(* CODESYS project bkp_29_07_24_VER_3_17.project
   Project Profile: Single

Project tree, tasks and I/O mapping:
  Device : NX3010, Altus S.A., order no. NX3010, version 1.2.1.233
    application Application
      libraries: NX5001 Diagnostic Structs, * (WAA); NX1005 Diagnostic Structs, * (WAA); NX2020 Diagnostic Structs, * (WAA); NX5000 Diagnostic Structs, * (WAA); NX6020 Diagnostic Structs, * (Manufacturer); Util, 3.5.1.0 (System); NextoStandard, 1.1.0.26 (WAA); LibDataTypes, 1.0.0.0 (Manufacturer); NX3010 Diagnostic Structs, 1.1.0.2 (WAA); NX2001 Diagnostic Structs, 1.0.0.5 (WAA); NX1001 Diagnostic Structs, 1.0.0.4 (WAA); NX6000 Diagnostic Structs, 0.0.0.2 (WAA); NX6010 Diagnostic Structs, 0.0.0.5 (Manufacturer); NX6100 Diagnostic Structs, 0.0.0.2 (WAA); NX4000 Diagnostic Structs, 1.0.0.0 (WAA); NXModbus Diagnostic Structs, 1.0.0.4 (WAA); NextoPID, 1.0.0.9 (WAA); Standard, 3.5.15.0 (System); Standard, * (System); SysTime, 3.5.9.0 (System); CAA File, 3.5.12.0 (CAA Technical Workgroup); CAA Callback Extern, 3.5.11.0 (CAA Technical Workgroup); CAA Memory Block Manager Extern, 3.5.7.0 (CAA Technical Workgroup); CAA Ressource Manager Extern, 3.5.11.0 (CAA Technical Workgroup); CAA Types Extern, 3.5.10.0 (CAA Technical Workgroup)
      task Configuration (cyclic, interval 9000 µs, priority 4) calls Configuration.EtherCAT_Task [Configuration.EtherCAT_Task]
      task MainTask (cyclic, interval 100 ms, priority 13, watchdog 1000 ms x 1) calls MainPrg
      task ATModbusMODBUS_Server (cyclic, interval 50 ms, priority 16) calls MODBUS_Server_Instance.Task
      task ATModbusMODBUS_RTU_Master (cyclic, interval 20 ms, priority 16) calls MODBUS_RTU_Master_Instance.Task
      Diagnostic Explorer
      Bill of Materials
      Configuration and Consumption
      program MainPrg [LD]
      global variables Diagnostics
      global variables PersistentVars
      global variables GVLStatus
      global variables GVLAlarmes
      global variables GVLGerais
      global variables GVLSlurryMaking
      program SlurryMaking [ST]
      program Transferencia [ST]
      global variables GVLTransferencia
      program Alarmes [ST]
      program FiltrosDeManga [ST]
      program SprayDrying [ST]
      global variables GVLTorre
      program PH [ST]
      global variables GVLPH
      program EA [ST]
      program SA [ST]
      global variables GVLTemperaturas
      program Temperturas [ST]
      global variables GVLSCHENCK
      program DSA1 [ST]
      program DSA2 [ST]
      program DSA3 [ST]
      program DSA4 [ST]
      program DSA5 [ST]
      program DSA7 [ST]
      program DSA8 [ST]
      program DSA9 [ST]
      program DSA10 [ST]
      program DSA11 [ST]
      program DSA12 [ST]
      program DSATorre [ST]
      program Status [ST]
      program DS6 [ST]
      program BBP01 [ST]
      program BBP02 [ST]
      program AutoPH [ST]
      global variables IOQualities
      trace Trace (task MainTask): Transferencia.PRESSAO_BOMBA, LEITURA_PRES_LB, PRST_PRESS_BB
      global variables Special_Variables
      program ProdL1 [ST]
      program ProdL2 [ST]
      program ProdL3 [ST]
      program ProdL4 [ST]
      program ProdL5 [ST]
      program ProdL6 [ST]
      program ProdL7 [ST]
      program ProdL8 [ST]
      program ProdL9 [ST]
      program ProdL10 [ST]
      program ProdAerossol [ST]
      program DSA14 [ST]
      global variables GVL_Ampliacao_transferencia
      program ampliacao_transferencia [ST]
      function block inv_modbus [ST]
    Configuration : Bus, WAA, order no. Configuration, version 1.1.1.2
        settings: MasterCycleTime = 4000
      NX3010 : NX3010, Altus S.A., order no. NX3010, version 1.2.1.233
          settings: DC sync0 cycletime = 4000; Generate Error if Task Whatchdog time greater than %80 of interval time = False; Consist retain and persistent area in %Q. = False; VFInitGenerate = False; Rack Configuration Info.Total Number of Racks = 2; Rack Configuration Info.Rack-0 Type = 9002; Rack Configuration Info.Rack-1 ID = 1; Rack Configuration Info.Rack-1 Type = 9002; IOModule's Address for interrupt = 255
        <Empty>
        COM 1
        COM 2
          MODBUS_RTU_Master : MODBUS RTU Master, WAA, version 1.0.0.8
              settings: Task Name = 'ATModbusMODBUS_RTU_Master'
            Dosador1 : MODBUS Device, WAA, version 1.0.0.8
                unmapped channels: %QD4000 Mapping Disabling
              Dosador1_Mapping_000 : Holding Register, WAA, version 1.0.0.8
              Dosador1_Mapping_001 : Holding Register, WAA, version 1.0.0.8
              Dosador1_Mapping_002 : Holding Register, WAA, version 1.0.0.8
              Dosador1_Mapping_003 : Holding Register, WAA, version 1.0.0.8
              Dosador1_Mapping_004 : Holding Register, WAA, version 1.0.0.8
              Dosador1_Mapping_005 : Holding Register, WAA, version 1.0.0.8
              Dosador1_Mapping_006 : Holding Register, WAA, version 1.0.0.8
              Dosador1_Mapping_007 : Holding Register, WAA, version 1.0.0.8
              Dosador1_Mapping_008 : Holding Register, WAA, version 1.0.0.8
              Dosador1_Mapping_009 : Holding Register, WAA, version 1.0.0.8
            Dosador2 : MODBUS Device, WAA, version 1.0.0.8
                unmapped channels: %QD4010 Mapping Disabling
              Dosador2_Mapping_000 : Holding Register, WAA, version 1.0.0.8
              Dosador2_Mapping_001 : Holding Register, WAA, version 1.0.0.8
              Dosador2_Mapping_002 : Holding Register, WAA, version 1.0.0.8
              Dosador2_Mapping_003 : Holding Register, WAA, version 1.0.0.8
              Dosador2_Mapping_004 : Holding Register, WAA, version 1.0.0.8
              Dosador2_Mapping_005 : Holding Register, WAA, version 1.0.0.8
              Dosador2_Mapping_006 : Holding Register, WAA, version 1.0.0.8
              Dosador2_Mapping_007 : Holding Register, WAA, version 1.0.0.8
              Dosador2_Mapping_008 : Holding Register, WAA, version 1.0.0.8
              Dosador2_Mapping_009 : Holding Register, WAA, version 1.0.0.8
            Dosador3 : MODBUS Device, WAA, version 1.0.0.8
                unmapped channels: %QD4020 Mapping Disabling
              Dosador3_Mapping_000 : Holding Register, WAA, version 1.0.0.8
              Dosador3_Mapping_001 : Holding Register, WAA, version 1.0.0.8
              Dosador3_Mapping_002 : Holding Register, WAA, version 1.0.0.8
              Dosador3_Mapping_003 : Holding Register, WAA, version 1.0.0.8
              Dosador3_Mapping_004 : Holding Register, WAA, version 1.0.0.8
              Dosador3_Mapping_005 : Holding Register, WAA, version 1.0.0.8
              Dosador3_Mapping_006 : Holding Register, WAA, version 1.0.0.8
              Dosador3_Mapping_007 : Holding Register, WAA, version 1.0.0.8
              Dosador3_Mapping_008 : Holding Register, WAA, version 1.0.0.8
              Dosador3_Mapping_009 : Holding Register, WAA, version 1.0.0.8
            Dosador4 : MODBUS Device, WAA, version 1.0.0.8
                unmapped channels: %QD4030 Mapping Disabling
              Dosador4_Mapping_000 : Holding Register, WAA, version 1.0.0.8
              Dosador4_Mapping_001 : Holding Register, WAA, version 1.0.0.8
              Dosador4_Mapping_002 : Holding Register, WAA, version 1.0.0.8
              Dosador4_Mapping_003 : Holding Register, WAA, version 1.0.0.8
              Dosador4_Mapping_004 : Holding Register, WAA, version 1.0.0.8
              Dosador4_Mapping_005 : Holding Register, WAA, version 1.0.0.8
              Dosador4_Mapping_006 : Holding Register, WAA, version 1.0.0.8
              Dosador4_Mapping_007 : Holding Register, WAA, version 1.0.0.8
              Dosador4_Mapping_008 : Holding Register, WAA, version 1.0.0.8
              Dosador4_Mapping_009 : Holding Register, WAA, version 1.0.0.8
            Dosador5 : MODBUS Device, WAA, version 1.0.0.8
                unmapped channels: %QD4040 Mapping Disabling
              Dosador5_Mapping_000 : Holding Register, WAA, version 1.0.0.8
              Dosador5_Mapping_001 : Holding Register, WAA, version 1.0.0.8
              Dosador5_Mapping_002 : Holding Register, WAA, version 1.0.0.8
              Dosador5_Mapping_003 : Holding Register, WAA, version 1.0.0.8
              Dosador5_Mapping_004 : Holding Register, WAA, version 1.0.0.8
              Dosador5_Mapping_005 : Holding Register, WAA, version 1.0.0.8
              Dosador5_Mapping_006 : Holding Register, WAA, version 1.0.0.8
              Dosador5_Mapping_007 : Holding Register, WAA, version 1.0.0.8
              Dosador5_Mapping_008 : Holding Register, WAA, version 1.0.0.8
              Dosador5_Mapping_009 : Holding Register, WAA, version 1.0.0.8
            Dosador7 : MODBUS Device, WAA, version 1.0.0.8
                unmapped channels: %QD4050 Mapping Disabling
              Dosador7_Mapping_000 : Holding Register, WAA, version 1.0.0.8
              Dosador7_Mapping_001 : Holding Register, WAA, version 1.0.0.8
              Dosador7_Mapping_002 : Holding Register, WAA, version 1.0.0.8
              Dosador7_Mapping_003 : Holding Register, WAA, version 1.0.0.8
              Dosador7_Mapping_004 : Holding Register, WAA, version 1.0.0.8
              Dosador7_Mapping_005 : Holding Register, WAA, version 1.0.0.8
              Dosador7_Mapping_006 : Holding Register, WAA, version 1.0.0.8
              Dosador7_Mapping_007 : Holding Register, WAA, version 1.0.0.8
              Dosador7_Mapping_008 : Holding Register, WAA, version 1.0.0.8
              Dosador7_Mapping_009 : Holding Register, WAA, version 1.0.0.8
            Dosador9 : MODBUS Device, WAA, version 1.0.0.8
                unmapped channels: %QD4070 Mapping Disabling
              Dosador9_Mapping_000 : Holding Register, WAA, version 1.0.0.8
              Dosador9_Mapping_001 : Holding Register, WAA, version 1.0.0.8
              Dosador9_Mapping_002 : Holding Register, WAA, version 1.0.0.8
              Dosador9_Mapping_003 : Holding Register, WAA, version 1.0.0.8
              Dosador9_Mapping_004 : Holding Register, WAA, version 1.0.0.8
              Dosador9_Mapping_005 : Holding Register, WAA, version 1.0.0.8
              Dosador9_Mapping_006 : Holding Register, WAA, version 1.0.0.8
              Dosador9_Mapping_007 : Holding Register, WAA, version 1.0.0.8
              Dosador9_Mapping_008 : Holding Register, WAA, version 1.0.0.8
              Dosador9_Mapping_009 : Holding Register, WAA, version 1.0.0.8
            Dosador8 : MODBUS Device, WAA, version 1.0.0.8
                unmapped channels: %QD4060 Mapping Disabling
              Dosador8_Mapping_000 : Holding Register, WAA, version 1.0.0.8
              Dosador8_Mapping_001 : Holding Register, WAA, version 1.0.0.8
              Dosador8_Mapping_002 : Holding Register, WAA, version 1.0.0.8
              Dosador8_Mapping_003 : Holding Register, WAA, version 1.0.0.8
              Dosador8_Mapping_004 : Holding Register, WAA, version 1.0.0.8
              Dosador8_Mapping_005 : Holding Register, WAA, version 1.0.0.8
              Dosador8_Mapping_006 : Holding Register, WAA, version 1.0.0.8
              Dosador8_Mapping_007 : Holding Register, WAA, version 1.0.0.8
              Dosador8_Mapping_008 : Holding Register, WAA, version 1.0.0.8
              Dosador8_Mapping_009 : Holding Register, WAA, version 1.0.0.8
            Dosador10 : MODBUS Device, WAA, version 1.0.0.8
                unmapped channels: %QD4080 Mapping Disabling
              Dosador10_Mapping_000 : Holding Register, WAA, version 1.0.0.8
              Dosador10_Mapping_001 : Holding Register, WAA, version 1.0.0.8
              Dosador10_Mapping_002 : Holding Register, WAA, version 1.0.0.8
              Dosador10_Mapping_003 : Holding Register, WAA, version 1.0.0.8
              Dosador10_Mapping_004 : Holding Register, WAA, version 1.0.0.8
              Dosador10_Mapping_005 : Holding Register, WAA, version 1.0.0.8
              Dosador10_Mapping_006 : Holding Register, WAA, version 1.0.0.8
              Dosador10_Mapping_007 : Holding Register, WAA, version 1.0.0.8
              Dosador10_Mapping_008 : Holding Register, WAA, version 1.0.0.8
              Dosador10_Mapping_009 : Holding Register, WAA, version 1.0.0.8
            Dosador11 : MODBUS Device, WAA, version 1.0.0.8
                unmapped channels: %QD4090 Mapping Disabling
              Dosador11_Mapping_000 : Holding Register, WAA, version 1.0.0.8
              Dosador11_Mapping_001 : Holding Register, WAA, version 1.0.0.8
              Dosador11_Mapping_002 : Holding Register, WAA, version 1.0.0.8
              Dosador11_Mapping_003 : Holding Register, WAA, version 1.0.0.8
              Dosador11_Mapping_004 : Holding Register, WAA, version 1.0.0.8
              Dosador11_Mapping_005 : Holding Register, WAA, version 1.0.0.8
              Dosador11_Mapping_006 : Holding Register, WAA, version 1.0.0.8
              Dosador11_Mapping_007 : Holding Register, WAA, version 1.0.0.8
              Dosador11_Mapping_008 : Holding Register, WAA, version 1.0.0.8
              Dosador11_Mapping_009 : Holding Register, WAA, version 1.0.0.8
            Dosador12 : MODBUS Device, WAA, version 1.0.0.8
                unmapped channels: %QD4100 Mapping Disabling
              Dosador12_Mapping_000 : Holding Register, WAA, version 1.0.0.8
              Dosador12_Mapping_001 : Holding Register, WAA, version 1.0.0.8
              Dosador12_Mapping_002 : Holding Register, WAA, version 1.0.0.8
              Dosador12_Mapping_003 : Holding Register, WAA, version 1.0.0.8
              Dosador12_Mapping_004 : Holding Register, WAA, version 1.0.0.8
              Dosador12_Mapping_005 : Holding Register, WAA, version 1.0.0.8
              Dosador12_Mapping_006 : Holding Register, WAA, version 1.0.0.8
              Dosador12_Mapping_007 : Holding Register, WAA, version 1.0.0.8
              Dosador12_Mapping_008 : Holding Register, WAA, version 1.0.0.8
              Dosador12_Mapping_009 : Holding Register, WAA, version 1.0.0.8
            Dosador13 : MODBUS Device, WAA, version 1.0.0.8
                unmapped channels: %QD4120 Mapping Disabling
              Dosador13_Mapping_000 : Holding Register, WAA, version 1.0.0.8
              Dosador13_Mapping_001 : Holding Register, WAA, version 1.0.0.8
              Dosador13_Mapping_002 : Holding Register, WAA, version 1.0.0.8
              Dosador13_Mapping_003 : Holding Register, WAA, version 1.0.0.8
              Dosador13_Mapping_004 : Holding Register, WAA, version 1.0.0.8
              Dosador13_Mapping_005 : Holding Register, WAA, version 1.0.0.8
              Dosador13_Mapping_006 : Holding Register, WAA, version 1.0.0.8
              Dosador13_Mapping_007 : Holding Register, WAA, version 1.0.0.8
              Dosador13_Mapping_008 : Holding Register, WAA, version 1.0.0.8
              Dosador13_Mapping_009 : Holding Register, WAA, version 1.0.0.8
            Dosador14 : MODBUS Device, WAA, version 1.0.0.8
                unmapped channels: %QD4140 Mapping Disabling
              Dosador14_Mapping_000 : Holding Register, WAA, version 1.0.0.8
              Dosador14_Mapping_001 : Holding Register, WAA, version 1.0.0.8
              Dosador14_Mapping_002 : Holding Register, WAA, version 1.0.0.8
              Dosador14_Mapping_006 : Holding Register, WAA, version 1.0.0.8
              Dosador14_Mapping_007 : Holding Register, WAA, version 1.0.0.8
              Dosador14_Mapping_008 : Holding Register, WAA, version 1.0.0.8
              Dosador14_Mapping_009 : Holding Register, WAA, version 1.0.0.8
        NET 1
            settings: IP Address = [10, 0, 0, 110]; Gateway Address = [10, 0, 0, 1]
          MODBUS_Server : MODBUS Server, WAA, version 1.0.0.9
              settings: Task Name = 'ATModbusMODBUS_Server'
              unmapped channels: %QD4096 Mapping Disabling
            MODBUS_Server_Mapping_001 : Holding Register, WAA, version 1.0.0.9
            MODBUS_Server_Mapping_000 : Coil, WAA, version 1.0.0.9
            MODBUS_Server_Mapping_002 : Holding Register, WAA, version 1.0.0.9
            MODBUS_Server_Mapping_003 : Holding Register, WAA, version 1.0.0.9
            MODBUS_Server_Mapping_004 : Holding Register, WAA, version 1.0.0.9
            MODBUS_Server_Mapping_005 : Holding Register, WAA, version 1.0.0.9
            MODBUS_Server_Mapping_006 : Holding Register, WAA, version 1.0.0.9
            MODBUS_Server_Mapping_007 : Holding Register, WAA, version 1.0.0.9
            MODBUS_Server_Mapping_008 : Coil, WAA, version 1.0.0.9
          MODBUS_Symbol_Client : MODBUS Symbol Client, Altus S.A., version 1.0.0.31
              settings: Diagnostic Variable.BaseType = 28; Diagnostic Variable.Address = ADR(Diagnostics.DG_MODBUS_Symbol_Client); Diagnostic Variable.SizeInBits = 160; Diagnostic Variable.TotalSizeInBits = 160
            INVERSOR_BOMBA_ALTA_03 : MODBUS Device, Altus S.A., version 1.0.0.31
                settings: IP Address = [10, 0, 0, 150]; Mappings definition.Count = 2; Item_00000.Value Variable.BaseType = 4; Item_00000.Value Variable.Address = ADR(GVL_Ampliacao_transferencia.BA_03_INV_LEITURA); Item_00000.Value Variable.SizeInBits = 32; Item_00000.Value Variable.TotalSizeInBits = 32; Item_00001.Value Variable.BaseType = 4; Item_00001.Value Variable.Address = ADR(GVL_Ampliacao_transferencia.BA_03_INV_ESCRITA); Item_00001.Value Variable.SizeInBits = 32; Item_00001.Value Variable.TotalSizeInBits = 32; Requests definition.Count = 2
            INVERSOR_BOMBA_BAIXA_02 : MODBUS Device, Altus S.A., version 1.0.0.31
                settings: IP Address = [10, 0, 0, 151]; Mappings definition.Count = 2; Item_00000.Value Variable.BaseType = 4; Item_00000.Value Variable.Address = ADR(GVL_Ampliacao_transferencia.BB_02_INV_LEITURA); Item_00000.Value Variable.SizeInBits = 32; Item_00000.Value Variable.TotalSizeInBits = 32; Item_00001.Value Variable.BaseType = 4; Item_00001.Value Variable.Address = ADR(GVL_Ampliacao_transferencia.BB_02_INV_ESCRITA); Item_00001.Value Variable.SizeInBits = 32; Item_00001.Value Variable.TotalSizeInBits = 32; Requests definition.Count = 2
            INVERSOR_MOINHO_02 : MODBUS Device, Altus S.A., version 1.0.0.31
                settings: IP Address = [10, 0, 0, 152]; Mappings definition.Count = 2; Item_00000.Value Variable.BaseType = 4; Item_00000.Value Variable.Address = ADR(GVL_Ampliacao_transferencia.MH_02_INV_LEITURA); Item_00000.Value Variable.SizeInBits = 32; Item_00000.Value Variable.TotalSizeInBits = 32; Item_00001.Value Variable.BaseType = 4; Item_00001.Value Variable.Address = ADR(GVL_Ampliacao_transferencia.BB_02_INV_ESCRITA); Item_00001.Value Variable.SizeInBits = 32; Item_00001.Value Variable.TotalSizeInBits = 32; Requests definition.Count = 2
            INVEROSR_MOINHO_01 : MODBUS Device, Altus S.A., version 1.0.0.31
                settings: IP Address = [10, 0, 0, 150]; Mappings definition.Count = 2; Item_00000.Value Variable.BaseType = 4; Item_00000.Value Variable.Address = ADR(GVL_Ampliacao_transferencia.MH_01_INV_LEITURA); Item_00000.Value Variable.SizeInBits = 32; Item_00000.Value Variable.TotalSizeInBits = 32; Item_00001.Value Variable.BaseType = 4; Item_00001.Value Variable.Address = ADR(GVL_Ampliacao_transferencia.MH_01_INV_ESCRITA); Item_00001.Value Variable.SizeInBits = 32; Item_00001.Value Variable.TotalSizeInBits = 32; Requests definition.Count = 2
        NX8000 : NX8000, Altus S.A., order no. NX8000, version 1.0.1.4
            settings: DC sync0 cycletime = 4000; Diag Instance Id = 0
        NX2001 : NX2001, Altus S.A., order no. NX2001, version 1.2.0.10
            settings: Physical Address of the Slave = 11; DC sync0 cycletime = 4000; Diag Instance Id = 11; %Q Start Address of Module Diagnostics Area = 21544; Parameter list definition.Count = 16; Item_00000.Access Name.BaseType = 1; Item_00000.Access Name.Address = ADR(IoConfig_Globals_Mapping.SD_RPO1); Item_00000.Access Name.SizeInBits = 1; Item_00000.Access Name.TotalSizeInBits = 1; Item_00001.Access Name.BaseType = 1; Item_00001.Access Name.Address = ADR(IoConfig_Globals_Mapping.SD_RPO2); Item_00001.Access Name.BitOffset = 1; Item_00001.Access Name.SizeInBits = 1; Item_00001.Access Name.TotalSizeInBits = 1; Item_00002.Access Name.BaseType = 1; Item_00002.Access Name.Address = ADR(IoConfig_Globals_Mapping.SD_RPO3); Item_00002.Access Name.BitOffset = 2; Item_00002.Access Name.SizeInBits = 1; Item_00002.Access Name.TotalSizeInBits = 1; Item_00003.Access Name.BaseType = 1; Item_00003.Access Name.Address = ADR(IoConfig_Globals_Mapping.SD_RPO4); Item_00003.Access Name.BitOffset = 3; Item_00003.Access Name.SizeInBits = 1; Item_00003.Access Name.TotalSizeInBits = 1; Item_00004.Access Name.BaseType = 1; Item_00004.Access Name.Address = ADR(IoConfig_Globals_Mapping.SD_RPO5); Item_00004.Access Name.BitOffset = 4; Item_00004.Access Name.SizeInBits = 1; Item_00004.Access Name.TotalSizeInBits = 1; Item_00005.Access Name.BaseType = 1; Item_00005.Access Name.Address = ADR(IoConfig_Globals_Mapping.SD_R6); Item_00005.Access Name.BitOffset = 5; Item_00005.Access Name.SizeInBits = 1; Item_00005.Access Name.TotalSizeInBits = 1; Item_00006.Access Name.BaseType = 1; Item_00006.Access Name.Address = ADR(IoConfig_Globals_Mapping.SD_R7); Item_00006.Access Name.BitOffset = 6; Item_00006.Access Name.SizeInBits = 1; Item_00006.Access Name.TotalSizeInBits = 1; Item_00007.Access Name.BaseType = 1;
              Item_00007.Access Name.Address = ADR(IoConfig_Globals_Mapping.SD_BLS1); Item_00007.Access Name.BitOffset = 7; Item_00007.Access Name.SizeInBits = 1; Item_00007.Access Name.TotalSizeInBits = 1; Item_00008.Access Name.BaseType = 1; Item_00008.Access Name.Address = ADR(IoConfig_Globals_Mapping.SD_BLS2); Item_00008.Access Name.SizeInBits = 1; Item_00008.Access Name.TotalSizeInBits = 1; Item_00009.Access Name.BaseType = 1; Item_00009.Access Name.Address = ADR(IoConfig_Globals_Mapping.SD_BLS3); Item_00009.Access Name.BitOffset = 1; Item_00009.Access Name.SizeInBits = 1; Item_00009.Access Name.TotalSizeInBits = 1; Item_00010.Access Name.BaseType = 1; Item_00010.Access Name.Address = ADR(IoConfig_Globals_Mapping.SD_BLS4); Item_00010.Access Name.BitOffset = 2; Item_00010.Access Name.SizeInBits = 1; Item_00010.Access Name.TotalSizeInBits = 1; Item_00011.Access Name.BaseType = 1; Item_00011.Access Name.Address = ADR(IoConfig_Globals_Mapping.SD_BLS5); Item_00011.Access Name.BitOffset = 3; Item_00011.Access Name.SizeInBits = 1; Item_00011.Access Name.TotalSizeInBits = 1; Item_00012.Access Name.BaseType = 1; Item_00012.Access Name.Address = ADR(IoConfig_Globals_Mapping.SD_BLL1R); Item_00012.Access Name.BitOffset = 4; Item_00012.Access Name.SizeInBits = 1; Item_00012.Access Name.TotalSizeInBits = 1; Item_00013.Access Name.BaseType = 1; Item_00013.Access Name.Address = ADR(IoConfig_Globals_Mapping.SD_BLL1L); Item_00013.Access Name.BitOffset = 5; Item_00013.Access Name.SizeInBits = 1; Item_00013.Access Name.TotalSizeInBits = 1; Item_00014.Access Name.BaseType = 1; Item_00014.Access Name.Address = ADR(IoConfig_Globals_Mapping.SD_BLL1D); Item_00014.Access Name.BitOffset = 6; Item_00014.Access Name.SizeInBits = 1; Item_00014.Access Name.TotalSizeInBits = 1; Item_00015.Access Name.BaseType = 1; Item_00015.Access Name.Address = ADR(IoConfig_Globals_Mapping.SD_BLL2L);
              Item_00015.Access Name.BitOffset = 7; Item_00015.Access Name.SizeInBits = 1; Item_00015.Access Name.TotalSizeInBits = 1; Quality Variable Name.BaseType = 28; Quality Variable Name.Address = ADR(IOQualities.QUALITY_NX2001); Quality Variable Name.SizeInBits = 32; Quality Variable Name.TotalSizeInBits = 512
            output SD_RPO1 : BOOL  // Digital Outputs - Byte 0.Output 00
            output SD_RPO2 : BOOL  // Digital Outputs - Byte 0.Output 01
            output SD_RPO3 : BOOL  // Digital Outputs - Byte 0.Output 02
            output SD_RPO4 : BOOL  // Digital Outputs - Byte 0.Output 03
            output SD_RPO5 : BOOL  // Digital Outputs - Byte 0.Output 04
            output SD_R6 : BOOL  // Digital Outputs - Byte 0.Output 05
            output SD_R7 : BOOL  // Digital Outputs - Byte 0.Output 06
            output SD_BLS1 : BOOL  // Digital Outputs - Byte 0.Output 07
            output SD_BLS2 : BOOL  // Digital Outputs - Byte 1.Output 10
            output SD_BLS3 : BOOL  // Digital Outputs - Byte 1.Output 11
            output SD_BLS4 : BOOL  // Digital Outputs - Byte 1.Output 12
            output SD_BLS5 : BOOL  // Digital Outputs - Byte 1.Output 13
            output SD_BLL1R : BOOL  // Digital Outputs - Byte 1.Output 14
            output SD_BLL1L : BOOL  // Digital Outputs - Byte 1.Output 15
            output SD_BLL1D : BOOL  // Digital Outputs - Byte 1.Output 16
            output SD_BLL2L : BOOL  // Digital Outputs - Byte 1.Output 17
            unmapped channels: %QB0 Digital Outputs - Byte 0, %QB1 Digital Outputs - Byte 1
        NX2001_01 : NX2001, Altus S.A., order no. NX2001, version 1.2.0.10
            settings: Physical Address of the Slave = 12; DC sync0 cycletime = 4000; Diag Instance Id = 12; %Q Start Address of Module Diagnostics Area = 21548; Parameter list definition.Count = 16; Item_00000.Access Name.BaseType = 1; Item_00000.Access Name.Address = ADR(IoConfig_Globals_Mapping.SD_BLBA1); Item_00000.Access Name.SizeInBits = 1; Item_00000.Access Name.TotalSizeInBits = 1; Item_00001.Access Name.BaseType = 1; Item_00001.Access Name.Address = ADR(IoConfig_Globals_Mapping.SD_BLL2D); Item_00001.Access Name.BitOffset = 1; Item_00001.Access Name.SizeInBits = 1; Item_00001.Access Name.TotalSizeInBits = 1; Item_00002.Access Name.BaseType = 1; Item_00002.Access Name.Address = ADR(IoConfig_Globals_Mapping.SD_BLL3R); Item_00002.Access Name.BitOffset = 2; Item_00002.Access Name.SizeInBits = 1; Item_00002.Access Name.TotalSizeInBits = 1; Item_00003.Access Name.BaseType = 1; Item_00003.Access Name.Address = ADR(IoConfig_Globals_Mapping.SD_BLL3L); Item_00003.Access Name.BitOffset = 3; Item_00003.Access Name.SizeInBits = 1; Item_00003.Access Name.TotalSizeInBits = 1; Item_00004.Access Name.BaseType = 1; Item_00004.Access Name.Address = ADR(IoConfig_Globals_Mapping.SD_BLL3D); Item_00004.Access Name.BitOffset = 4; Item_00004.Access Name.SizeInBits = 1; Item_00004.Access Name.TotalSizeInBits = 1; Item_00005.Access Name.BaseType = 1; Item_00005.Access Name.Address = ADR(IoConfig_Globals_Mapping.SD_BLL4R); Item_00005.Access Name.BitOffset = 5; Item_00005.Access Name.SizeInBits = 1; Item_00005.Access Name.TotalSizeInBits = 1; Item_00006.Access Name.BaseType = 1; Item_00006.Access Name.Address = ADR(IoConfig_Globals_Mapping.SD_BLL4L); Item_00006.Access Name.BitOffset = 6; Item_00006.Access Name.SizeInBits = 1; Item_00006.Access Name.TotalSizeInBits = 1; Item_00007.Access Name.BaseType = 1;
              Item_00007.Access Name.Address = ADR(IoConfig_Globals_Mapping.SD_BLL4D); Item_00007.Access Name.BitOffset = 7; Item_00007.Access Name.SizeInBits = 1; Item_00007.Access Name.TotalSizeInBits = 1; Item_00008.Access Name.BaseType = 1; Item_00008.Access Name.Address = ADR(IoConfig_Globals_Mapping.SD_MXP_P); Item_00008.Access Name.SizeInBits = 1; Item_00008.Access Name.TotalSizeInBits = 1; Item_00009.Access Name.BaseType = 1; Item_00009.Access Name.Address = ADR(IoConfig_Globals_Mapping.SD_MXP_E); Item_00009.Access Name.BitOffset = 1; Item_00009.Access Name.SizeInBits = 1; Item_00009.Access Name.TotalSizeInBits = 1; Item_00010.Access Name.BaseType = 1; Item_00010.Access Name.Address = ADR(IoConfig_Globals_Mapping.SD_MXP_T); Item_00010.Access Name.BitOffset = 2; Item_00010.Access Name.SizeInBits = 1; Item_00010.Access Name.TotalSizeInBits = 1; Item_00011.Access Name.BaseType = 1; Item_00011.Access Name.Address = ADR(IoConfig_Globals_Mapping.SD_VPMECEDOR); Item_00011.Access Name.BitOffset = 3; Item_00011.Access Name.SizeInBits = 1; Item_00011.Access Name.TotalSizeInBits = 1; Item_00012.Access Name.BaseType = 1; Item_00012.Access Name.Address = ADR(IoConfig_Globals_Mapping.BL_03_CMD); Item_00012.Access Name.BitOffset = 4; Item_00012.Access Name.SizeInBits = 1; Item_00012.Access Name.TotalSizeInBits = 1; Item_00013.Access Name.BaseType = 1; Item_00013.Access Name.Address = ADR(IoConfig_Globals_Mapping.SD_MH_E); Item_00013.Access Name.BitOffset = 5; Item_00013.Access Name.SizeInBits = 1; Item_00013.Access Name.TotalSizeInBits = 1; Item_00014.Access Name.BaseType = 1; Item_00014.Access Name.Address = ADR(IoConfig_Globals_Mapping.SD_MH_T); Item_00014.Access Name.BitOffset = 6; Item_00014.Access Name.SizeInBits = 1; Item_00014.Access Name.TotalSizeInBits = 1; Item_00015.Access Name.BaseType = 1; Item_00015.Access Name.Address = ADR(IoConfig_Globals_Mapping.SD_MXESPERA);
              Item_00015.Access Name.BitOffset = 7; Item_00015.Access Name.SizeInBits = 1; Item_00015.Access Name.TotalSizeInBits = 1; Quality Variable Name.BaseType = 28; Quality Variable Name.Address = ADR(IOQualities.QUALITY_NX2001_01); Quality Variable Name.SizeInBits = 32; Quality Variable Name.TotalSizeInBits = 512
            output SD_BLBA1 : BOOL  // Digital Outputs - Byte 0.Output 00
            output SD_BLL2D : BOOL  // Digital Outputs - Byte 0.Output 01
            output SD_BLL3R : BOOL  // Digital Outputs - Byte 0.Output 02
            output SD_BLL3L : BOOL  // Digital Outputs - Byte 0.Output 03
            output SD_BLL3D : BOOL  // Digital Outputs - Byte 0.Output 04
            output SD_BLL4R : BOOL  // Digital Outputs - Byte 0.Output 05
            output SD_BLL4L : BOOL  // Digital Outputs - Byte 0.Output 06
            output SD_BLL4D : BOOL  // Digital Outputs - Byte 0.Output 07
            output SD_MXP_P : BOOL  // Digital Outputs - Byte 1.Output 10
            output SD_MXP_E : BOOL  // Digital Outputs - Byte 1.Output 11
            output SD_MXP_T : BOOL  // Digital Outputs - Byte 1.Output 12
            output SD_VPMECEDOR : BOOL  // Digital Outputs - Byte 1.Output 13
            output BL_03_CMD : BOOL  // Digital Outputs - Byte 1.Output 14
            output SD_MH_E : BOOL  // Digital Outputs - Byte 1.Output 15
            output SD_MH_T : BOOL  // Digital Outputs - Byte 1.Output 16
            output SD_MXESPERA : BOOL  // Digital Outputs - Byte 1.Output 17
            unmapped channels: %QB2 Digital Outputs - Byte 0, %QB3 Digital Outputs - Byte 1
        NX2001_02 : NX2001, Altus S.A., order no. NX2001, version 1.2.0.10
            settings: Physical Address of the Slave = 13; DC sync0 cycletime = 4000; Diag Instance Id = 13; %Q Start Address of Module Diagnostics Area = 21552; Parameter list definition.Count = 16; Item_00000.Access Name.BaseType = 1; Item_00000.Access Name.Address = ADR(IoConfig_Globals_Mapping.SD_BSUL); Item_00000.Access Name.SizeInBits = 1; Item_00000.Access Name.TotalSizeInBits = 1; Item_00001.Access Name.BaseType = 1; Item_00001.Access Name.Address = ADR(IoConfig_Globals_Mapping.SD_BSIL); Item_00001.Access Name.BitOffset = 1; Item_00001.Access Name.SizeInBits = 1; Item_00001.Access Name.TotalSizeInBits = 1; Item_00002.Access Name.BaseType = 1; Item_00002.Access Name.Address = ADR(IoConfig_Globals_Mapping.SD_BAG); Item_00002.Access Name.BitOffset = 2; Item_00002.Access Name.SizeInBits = 1; Item_00002.Access Name.TotalSizeInBits = 1; Item_00003.Access Name.BaseType = 1; Item_00003.Access Name.Address = ADR(IoConfig_Globals_Mapping.SD_BBD); Item_00003.Access Name.BitOffset = 3; Item_00003.Access Name.SizeInBits = 1; Item_00003.Access Name.TotalSizeInBits = 1; Item_00004.Access Name.BaseType = 1; Item_00004.Access Name.Address = ADR(IoConfig_Globals_Mapping.SD_BBTRANS); Item_00004.Access Name.BitOffset = 4; Item_00004.Access Name.SizeInBits = 1; Item_00004.Access Name.TotalSizeInBits = 1; Item_00005.Access Name.BaseType = 1; Item_00005.Access Name.Address = ADR(IoConfig_Globals_Mapping.SD_BB); Item_00005.Access Name.BitOffset = 5; Item_00005.Access Name.SizeInBits = 1; Item_00005.Access Name.TotalSizeInBits = 1; Item_00006.Access Name.BaseType = 1; Item_00006.Access Name.Address = ADR(IoConfig_Globals_Mapping.SD_BA1); Item_00006.Access Name.BitOffset = 6; Item_00006.Access Name.SizeInBits = 1; Item_00006.Access Name.TotalSizeInBits = 1; Item_00007.Access Name.BaseType = 1;
              Item_00007.Access Name.Address = ADR(IoConfig_Globals_Mapping.SD_BA2); Item_00007.Access Name.BitOffset = 7; Item_00007.Access Name.SizeInBits = 1; Item_00007.Access Name.TotalSizeInBits = 1; Item_00008.Access Name.BaseType = 1; Item_00008.Access Name.Address = ADR(IoConfig_Globals_Mapping.AL_SIR_DOSADORES); Item_00008.Access Name.SizeInBits = 1; Item_00008.Access Name.TotalSizeInBits = 1; Item_00009.Access Name.BaseType = 1; Item_00009.Access Name.Address = ADR(IoConfig_Globals_Mapping.SD_BSOD); Item_00009.Access Name.BitOffset = 1; Item_00009.Access Name.SizeInBits = 1; Item_00009.Access Name.TotalSizeInBits = 1; Item_00010.Access Name.BaseType = 1; Item_00010.Access Name.Address = ADR(IoConfig_Globals_Mapping.SD_BACU); Item_00010.Access Name.BitOffset = 2; Item_00010.Access Name.SizeInBits = 1; Item_00010.Access Name.TotalSizeInBits = 1; Item_00011.Access Name.BaseType = 1; Item_00011.Access Name.Address = ADR(IoConfig_Globals_Mapping.SD_BPER1); Item_00011.Access Name.BitOffset = 3; Item_00011.Access Name.SizeInBits = 1; Item_00011.Access Name.TotalSizeInBits = 1; Item_00012.Access Name.BaseType = 1; Item_00012.Access Name.Address = ADR(IoConfig_Globals_Mapping.SD_BPER2); Item_00012.Access Name.BitOffset = 4; Item_00012.Access Name.SizeInBits = 1; Item_00012.Access Name.TotalSizeInBits = 1; Item_00013.Access Name.BaseType = 1; Item_00013.Access Name.Address = ADR(IoConfig_Globals_Mapping.SD_RoscaCelquim); Item_00013.Access Name.BitOffset = 5; Item_00013.Access Name.SizeInBits = 1; Item_00013.Access Name.TotalSizeInBits = 1; Item_00014.Access Name.BaseType = 1; Item_00014.Access Name.Address = ADR(IoConfig_Globals_Mapping.SD_BAO); Item_00014.Access Name.BitOffset = 6; Item_00014.Access Name.SizeInBits = 1; Item_00014.Access Name.TotalSizeInBits = 1; Item_00015.Access Name.BaseType = 1; Item_00015.Access Name.Address = ADR(IoConfig_Globals_Mapping.SD_BLBA2);
              Item_00015.Access Name.BitOffset = 7; Item_00015.Access Name.SizeInBits = 1; Item_00015.Access Name.TotalSizeInBits = 1; Quality Variable Name.BaseType = 28; Quality Variable Name.Address = ADR(IOQualities.QUALITY_NX2001_02); Quality Variable Name.SizeInBits = 32; Quality Variable Name.TotalSizeInBits = 512
            output SD_BSUL : BOOL  // Digital Outputs - Byte 0.Output 00
            output SD_BSIL : BOOL  // Digital Outputs - Byte 0.Output 01
            output SD_BAG : BOOL  // Digital Outputs - Byte 0.Output 02
            output SD_BBD : BOOL  // Digital Outputs - Byte 0.Output 03
            output SD_BBTRANS : BOOL  // Digital Outputs - Byte 0.Output 04
            output SD_BB : BOOL  // Digital Outputs - Byte 0.Output 05
            output SD_BA1 : BOOL  // Digital Outputs - Byte 0.Output 06
            output SD_BA2 : BOOL  // Digital Outputs - Byte 0.Output 07
            output AL_SIR_DOSADORES : BOOL  // Digital Outputs - Byte 1.Output 10
            output SD_BSOD : BOOL  // Digital Outputs - Byte 1.Output 11
            output SD_BACU : BOOL  // Digital Outputs - Byte 1.Output 12
            output SD_BPER1 : BOOL  // Digital Outputs - Byte 1.Output 13
            output SD_BPER2 : BOOL  // Digital Outputs - Byte 1.Output 14
            output SD_RoscaCelquim : BOOL  // Digital Outputs - Byte 1.Output 15
            output SD_BAO : BOOL  // Digital Outputs - Byte 1.Output 16
            output SD_BLBA2 : BOOL  // Digital Outputs - Byte 1.Output 17
            unmapped channels: %QB4 Digital Outputs - Byte 0, %QB5 Digital Outputs - Byte 1
        NX2001_03 : NX2001, Altus S.A., order no. NX2001, version 1.2.0.10
            settings: Physical Address of the Slave = 258; DC sync0 cycletime = 4000; Diag Instance Id = 258; %Q Start Address of Module Diagnostics Area = 21556; Parameter list definition.Count = 16; Item_00000.Access Name.BaseType = 1; Item_00000.Access Name.Address = ADR(IoConfig_Globals_Mapping.SD_VLMISTURA); Item_00000.Access Name.SizeInBits = 1; Item_00000.Access Name.TotalSizeInBits = 1; Item_00001.Access Name.BaseType = 1; Item_00001.Access Name.Address = ADR(IoConfig_Globals_Mapping.SD_VLR); Item_00001.Access Name.BitOffset = 1; Item_00001.Access Name.SizeInBits = 1; Item_00001.Access Name.TotalSizeInBits = 1; Item_00002.Access Name.BaseType = 1; Item_00002.Access Name.Address = ADR(IoConfig_Globals_Mapping.SD_VLAG); Item_00002.Access Name.BitOffset = 2; Item_00002.Access Name.SizeInBits = 1; Item_00002.Access Name.TotalSizeInBits = 1; Item_00003.Access Name.BaseType = 1; Item_00003.Access Name.Address = ADR(IoConfig_Globals_Mapping.SD_VLACU); Item_00003.Access Name.BitOffset = 3; Item_00003.Access Name.SizeInBits = 1; Item_00003.Access Name.TotalSizeInBits = 1; Item_00004.Access Name.BaseType = 1; Item_00004.Access Name.Address = ADR(IoConfig_Globals_Mapping.SD_FLT11); Item_00004.Access Name.BitOffset = 4; Item_00004.Access Name.SizeInBits = 1; Item_00004.Access Name.TotalSizeInBits = 1; Item_00005.Access Name.BaseType = 1; Item_00005.Access Name.Address = ADR(IoConfig_Globals_Mapping.SD_FLT12); Item_00005.Access Name.BitOffset = 5; Item_00005.Access Name.SizeInBits = 1; Item_00005.Access Name.TotalSizeInBits = 1; Item_00006.Access Name.BaseType = 1; Item_00006.Access Name.Address = ADR(IoConfig_Globals_Mapping.SD_FLT13); Item_00006.Access Name.BitOffset = 6; Item_00006.Access Name.SizeInBits = 1; Item_00006.Access Name.TotalSizeInBits = 1; Item_00007.Access Name.BaseType = 1;
              Item_00007.Access Name.Address = ADR(IoConfig_Globals_Mapping.SD_FLT14); Item_00007.Access Name.BitOffset = 7; Item_00007.Access Name.SizeInBits = 1; Item_00007.Access Name.TotalSizeInBits = 1; Item_00008.Access Name.BaseType = 1; Item_00008.Access Name.Address = ADR(IoConfig_Globals_Mapping.SD_FILT2123); Item_00008.Access Name.SizeInBits = 1; Item_00008.Access Name.TotalSizeInBits = 1; Item_00009.Access Name.BaseType = 1; Item_00009.Access Name.Address = ADR(IoConfig_Globals_Mapping.SD_FILT2224); Item_00009.Access Name.BitOffset = 1; Item_00009.Access Name.SizeInBits = 1; Item_00009.Access Name.TotalSizeInBits = 1; Item_00010.Access Name.BaseType = 1; Item_00010.Access Name.Address = ADR(IoConfig_Globals_Mapping.SD_FILT3133); Item_00010.Access Name.BitOffset = 2; Item_00010.Access Name.SizeInBits = 1; Item_00010.Access Name.TotalSizeInBits = 1; Item_00011.Access Name.BaseType = 1; Item_00011.Access Name.Address = ADR(IoConfig_Globals_Mapping.SD_FILT3234); Item_00011.Access Name.BitOffset = 3; Item_00011.Access Name.SizeInBits = 1; Item_00011.Access Name.TotalSizeInBits = 1; Item_00012.Access Name.BaseType = 1; Item_00012.Access Name.Address = ADR(IoConfig_Globals_Mapping.SD_EXFM1_P); Item_00012.Access Name.BitOffset = 4; Item_00012.Access Name.SizeInBits = 1; Item_00012.Access Name.TotalSizeInBits = 1; Item_00013.Access Name.BaseType = 1; Item_00013.Access Name.Address = ADR(IoConfig_Globals_Mapping.SD_EXFM1_E); Item_00013.Access Name.BitOffset = 5; Item_00013.Access Name.SizeInBits = 1; Item_00013.Access Name.TotalSizeInBits = 1; Item_00014.Access Name.BaseType = 1; Item_00014.Access Name.Address = ADR(IoConfig_Globals_Mapping.SD_EXFM1_T); Item_00014.Access Name.BitOffset = 6; Item_00014.Access Name.SizeInBits = 1; Item_00014.Access Name.TotalSizeInBits = 1; Item_00015.Access Name.BaseType = 1; Item_00015.Access Name.Address = ADR(IoConfig_Globals_Mapping.SD_EXFM2_P);
              Item_00015.Access Name.BitOffset = 7; Item_00015.Access Name.SizeInBits = 1; Item_00015.Access Name.TotalSizeInBits = 1; Quality Variable Name.BaseType = 28; Quality Variable Name.Address = ADR(IOQualities.QUALITY_NX2001_03); Quality Variable Name.SizeInBits = 32; Quality Variable Name.TotalSizeInBits = 512
            output SD_VLMISTURA : BOOL  // Digital Outputs - Byte 0.Output 00
            output SD_VLR : BOOL  // Digital Outputs - Byte 0.Output 01
            output SD_VLAG : BOOL  // Digital Outputs - Byte 0.Output 02
            output SD_VLACU : BOOL  // Digital Outputs - Byte 0.Output 03
            output SD_FLT11 : BOOL  // Digital Outputs - Byte 0.Output 04
            output SD_FLT12 : BOOL  // Digital Outputs - Byte 0.Output 05
            output SD_FLT13 : BOOL  // Digital Outputs - Byte 0.Output 06
            output SD_FLT14 : BOOL  // Digital Outputs - Byte 0.Output 07
            output SD_FILT2123 : BOOL  // Digital Outputs - Byte 1.Output 10
            output SD_FILT2224 : BOOL  // Digital Outputs - Byte 1.Output 11
            output SD_FILT3133 : BOOL  // Digital Outputs - Byte 1.Output 12
            output SD_FILT3234 : BOOL  // Digital Outputs - Byte 1.Output 13
            output SD_EXFM1_P : BOOL  // Digital Outputs - Byte 1.Output 14
            output SD_EXFM1_E : BOOL  // Digital Outputs - Byte 1.Output 15
            output SD_EXFM1_T : BOOL  // Digital Outputs - Byte 1.Output 16
            output SD_EXFM2_P : BOOL  // Digital Outputs - Byte 1.Output 17
            unmapped channels: %QB6 Digital Outputs - Byte 0, %QB7 Digital Outputs - Byte 1
        NX2001_04 : NX2001, Altus S.A., order no. NX2001, version 1.2.0.10
            settings: Physical Address of the Slave = 259; DC sync0 cycletime = 4000; Diag Instance Id = 259; %Q Start Address of Module Diagnostics Area = 21560; Parameter list definition.Count = 16; Item_00000.Access Name.BaseType = 1; Item_00000.Access Name.Address = ADR(IoConfig_Globals_Mapping.SD_EXFM2_E); Item_00000.Access Name.SizeInBits = 1; Item_00000.Access Name.TotalSizeInBits = 1; Item_00001.Access Name.BaseType = 1; Item_00001.Access Name.Address = ADR(IoConfig_Globals_Mapping.SD_EXFM2_T); Item_00001.Access Name.BitOffset = 1; Item_00001.Access Name.SizeInBits = 1; Item_00001.Access Name.TotalSizeInBits = 1; Item_00002.Access Name.BaseType = 1; Item_00002.Access Name.Address = ADR(IoConfig_Globals_Mapping.SD_VEXFM2_P); Item_00002.Access Name.BitOffset = 2; Item_00002.Access Name.SizeInBits = 1; Item_00002.Access Name.TotalSizeInBits = 1; Item_00003.Access Name.BaseType = 1; Item_00003.Access Name.Address = ADR(IoConfig_Globals_Mapping.SD_VEXFM2_E); Item_00003.Access Name.BitOffset = 3; Item_00003.Access Name.SizeInBits = 1; Item_00003.Access Name.TotalSizeInBits = 1; Item_00004.Access Name.BaseType = 1; Item_00004.Access Name.Address = ADR(IoConfig_Globals_Mapping.SD_VEXFM2_T); Item_00004.Access Name.BitOffset = 4; Item_00004.Access Name.SizeInBits = 1; Item_00004.Access Name.TotalSizeInBits = 1; Item_00005.Access Name.BaseType = 1; Item_00005.Access Name.Address = ADR(IoConfig_Globals_Mapping.SD_EX125); Item_00005.Access Name.BitOffset = 5; Item_00005.Access Name.SizeInBits = 1; Item_00005.Access Name.TotalSizeInBits = 1; Item_00006.Access Name.BaseType = 1; Item_00006.Access Name.Address = ADR(IoConfig_Globals_Mapping.SD_EX100); Item_00006.Access Name.BitOffset = 6; Item_00006.Access Name.SizeInBits = 1; Item_00006.Access Name.TotalSizeInBits = 1; Item_00007.Access Name.BaseType = 1;
              Item_00007.Access Name.Address = ADR(IoConfig_Globals_Mapping.SD_VFLU); Item_00007.Access Name.BitOffset = 7; Item_00007.Access Name.SizeInBits = 1; Item_00007.Access Name.TotalSizeInBits = 1; Item_00008.Access Name.BaseType = 1; Item_00008.Access Name.Address = ADR(IoConfig_Globals_Mapping.SD_ESTTC3); Item_00008.Access Name.SizeInBits = 1; Item_00008.Access Name.TotalSizeInBits = 1; Item_00009.Access Name.BaseType = 1; Item_00009.Access Name.Address = ADR(IoConfig_Globals_Mapping.SD_ESTPOB1); Item_00009.Access Name.BitOffset = 1; Item_00009.Access Name.SizeInBits = 1; Item_00009.Access Name.TotalSizeInBits = 1; Item_00010.Access Name.BaseType = 1; Item_00010.Access Name.Address = ADR(IoConfig_Globals_Mapping.SD_ESTPOB1_R); Item_00010.Access Name.BitOffset = 2; Item_00010.Access Name.SizeInBits = 1; Item_00010.Access Name.TotalSizeInBits = 1; Item_00011.Access Name.BaseType = 1; Item_00011.Access Name.Address = ADR(IoConfig_Globals_Mapping.SD_ESTTC8); Item_00011.Access Name.BitOffset = 3; Item_00011.Access Name.SizeInBits = 1; Item_00011.Access Name.TotalSizeInBits = 1; Item_00012.Access Name.BaseType = 1; Item_00012.Access Name.Address = ADR(IoConfig_Globals_Mapping.SD_ESTTC8_R); Item_00012.Access Name.BitOffset = 4; Item_00012.Access Name.SizeInBits = 1; Item_00012.Access Name.TotalSizeInBits = 1; Item_00013.Access Name.BaseType = 1; Item_00013.Access Name.Address = ADR(IoConfig_Globals_Mapping.SD_ESTTC9); Item_00013.Access Name.BitOffset = 5; Item_00013.Access Name.SizeInBits = 1; Item_00013.Access Name.TotalSizeInBits = 1; Item_00014.Access Name.BaseType = 1; Item_00014.Access Name.Address = ADR(IoConfig_Globals_Mapping.SD_ESTTC10); Item_00014.Access Name.BitOffset = 6; Item_00014.Access Name.SizeInBits = 1; Item_00014.Access Name.TotalSizeInBits = 1; Item_00015.Access Name.BaseType = 1; Item_00015.Access Name.Address = ADR(IoConfig_Globals_Mapping.SD_ESTPOB11);
              Item_00015.Access Name.BitOffset = 7; Item_00015.Access Name.SizeInBits = 1; Item_00015.Access Name.TotalSizeInBits = 1; Quality Variable Name.BaseType = 28; Quality Variable Name.Address = ADR(IOQualities.QUALITY_NX2001_04); Quality Variable Name.SizeInBits = 32; Quality Variable Name.TotalSizeInBits = 512
            output SD_EXFM2_E : BOOL  // Digital Outputs - Byte 0.Output 00
            output SD_EXFM2_T : BOOL  // Digital Outputs - Byte 0.Output 01
            output SD_VEXFM2_P : BOOL  // Digital Outputs - Byte 0.Output 02
            output SD_VEXFM2_E : BOOL  // Digital Outputs - Byte 0.Output 03
            output SD_VEXFM2_T : BOOL  // Digital Outputs - Byte 0.Output 04
            output SD_EX125 : BOOL  // Digital Outputs - Byte 0.Output 05
            output SD_EX100 : BOOL  // Digital Outputs - Byte 0.Output 06
            output SD_VFLU : BOOL  // Digital Outputs - Byte 0.Output 07
            output SD_ESTTC3 : BOOL  // Digital Outputs - Byte 1.Output 10
            output SD_ESTPOB1 : BOOL  // Digital Outputs - Byte 1.Output 11
            output SD_ESTPOB1_R : BOOL  // Digital Outputs - Byte 1.Output 12
            output SD_ESTTC8 : BOOL  // Digital Outputs - Byte 1.Output 13
            output SD_ESTTC8_R : BOOL  // Digital Outputs - Byte 1.Output 14
            output SD_ESTTC9 : BOOL  // Digital Outputs - Byte 1.Output 15
            output SD_ESTTC10 : BOOL  // Digital Outputs - Byte 1.Output 16
            output SD_ESTPOB11 : BOOL  // Digital Outputs - Byte 1.Output 17
            unmapped channels: %QB8 Digital Outputs - Byte 0, %QB9 Digital Outputs - Byte 1
        NX2001_05 : NX2001, Altus S.A., order no. NX2001, version 1.2.0.10
            settings: Physical Address of the Slave = 260; DC sync0 cycletime = 4000; Diag Instance Id = 260; %Q Start Address of Module Diagnostics Area = 21564; Parameter list definition.Count = 16; Item_00000.Access Name.BaseType = 1; Item_00000.Access Name.Address = ADR(IoConfig_Globals_Mapping.SD_ESTTC02); Item_00000.Access Name.SizeInBits = 1; Item_00000.Access Name.TotalSizeInBits = 1; Item_00001.Access Name.BaseType = 1; Item_00001.Access Name.Address = ADR(IoConfig_Globals_Mapping.SD_ESTTC12); Item_00001.Access Name.BitOffset = 1; Item_00001.Access Name.SizeInBits = 1; Item_00001.Access Name.TotalSizeInBits = 1; Item_00002.Access Name.BaseType = 1; Item_00002.Access Name.Address = ADR(IoConfig_Globals_Mapping.SD_ESTTC13); Item_00002.Access Name.BitOffset = 2; Item_00002.Access Name.SizeInBits = 1; Item_00002.Access Name.TotalSizeInBits = 1; Item_00003.Access Name.BaseType = 1; Item_00003.Access Name.Address = ADR(IoConfig_Globals_Mapping.SD_ESTSTORRE); Item_00003.Access Name.BitOffset = 3; Item_00003.Access Name.SizeInBits = 1; Item_00003.Access Name.TotalSizeInBits = 1; Item_00004.Access Name.BaseType = 1; Item_00004.Access Name.Address = ADR(IoConfig_Globals_Mapping.SD_ESTDSSUL); Item_00004.Access Name.BitOffset = 4; Item_00004.Access Name.SizeInBits = 1; Item_00004.Access Name.TotalSizeInBits = 1; Item_00005.Access Name.BaseType = 1; Item_00005.Access Name.Address = ADR(IoConfig_Globals_Mapping.SD_ESTSAIRLIF); Item_00005.Access Name.BitOffset = 5; Item_00005.Access Name.SizeInBits = 1; Item_00005.Access Name.TotalSizeInBits = 1; Item_00006.Access Name.BaseType = 1; Item_00006.Access Name.Address = ADR(IoConfig_Globals_Mapping.SD_DS6); Item_00006.Access Name.BitOffset = 6; Item_00006.Access Name.SizeInBits = 1; Item_00006.Access Name.TotalSizeInBits = 1; Item_00007.Access Name.BaseType = 1;
              Item_00007.Access Name.Address = ADR(IoConfig_Globals_Mapping.SD_DSASULTOR); Item_00007.Access Name.BitOffset = 7; Item_00007.Access Name.SizeInBits = 1; Item_00007.Access Name.TotalSizeInBits = 1; Item_00008.Access Name.BaseType = 1; Item_00008.Access Name.Address = ADR(IoConfig_Globals_Mapping.SD_EL2DMIX); Item_00008.Access Name.SizeInBits = 1; Item_00008.Access Name.TotalSizeInBits = 1; Item_00009.Access Name.BaseType = 1; Item_00009.Access Name.Address = ADR(IoConfig_Globals_Mapping.SD_EL2); Item_00009.Access Name.BitOffset = 1; Item_00009.Access Name.SizeInBits = 1; Item_00009.Access Name.TotalSizeInBits = 1; Item_00010.Access Name.BaseType = 1; Item_00010.Access Name.Address = ADR(IoConfig_Globals_Mapping.SD_M1PN); Item_00010.Access Name.BitOffset = 2; Item_00010.Access Name.SizeInBits = 1; Item_00010.Access Name.TotalSizeInBits = 1; Item_00011.Access Name.BaseType = 1; Item_00011.Access Name.Address = ADR(IoConfig_Globals_Mapping.SD_M2PN); Item_00011.Access Name.BitOffset = 3; Item_00011.Access Name.SizeInBits = 1; Item_00011.Access Name.TotalSizeInBits = 1; Item_00012.Access Name.BaseType = 1; Item_00012.Access Name.Address = ADR(IoConfig_Globals_Mapping.SD_M3PN); Item_00012.Access Name.BitOffset = 4; Item_00012.Access Name.SizeInBits = 1; Item_00012.Access Name.TotalSizeInBits = 1; Item_00013.Access Name.BaseType = 1; Item_00013.Access Name.Address = ADR(IoConfig_Globals_Mapping.SD_M4PN); Item_00013.Access Name.BitOffset = 5; Item_00013.Access Name.SizeInBits = 1; Item_00013.Access Name.TotalSizeInBits = 1; Item_00014.Access Name.BaseType = 1; Item_00014.Access Name.Address = ADR(IoConfig_Globals_Mapping.SD_LQUEI); Item_00014.Access Name.BitOffset = 6; Item_00014.Access Name.SizeInBits = 1; Item_00014.Access Name.TotalSizeInBits = 1; Item_00015.Access Name.BaseType = 1; Item_00015.Access Name.Address = ADR(IoConfig_Globals_Mapping.SD_MAIRLIF);
              Item_00015.Access Name.BitOffset = 7; Item_00015.Access Name.SizeInBits = 1; Item_00015.Access Name.TotalSizeInBits = 1; Quality Variable Name.BaseType = 28; Quality Variable Name.Address = ADR(IOQualities.QUALITY_NX2001_05); Quality Variable Name.SizeInBits = 32; Quality Variable Name.TotalSizeInBits = 512
            output SD_ESTTC02 : BOOL  // Digital Outputs - Byte 0.Output 00
            output SD_ESTTC12 : BOOL  // Digital Outputs - Byte 0.Output 01
            output SD_ESTTC13 : BOOL  // Digital Outputs - Byte 0.Output 02
            output SD_ESTSTORRE : BOOL  // Digital Outputs - Byte 0.Output 03
            output SD_ESTDSSUL : BOOL  // Digital Outputs - Byte 0.Output 04
            output SD_ESTSAIRLIF : BOOL  // Digital Outputs - Byte 0.Output 05
            output SD_DS6 : BOOL  // Digital Outputs - Byte 0.Output 06
            output SD_DSASULTOR : BOOL  // Digital Outputs - Byte 0.Output 07
            output SD_EL2DMIX : BOOL  // Digital Outputs - Byte 1.Output 10
            output SD_EL2 : BOOL  // Digital Outputs - Byte 1.Output 11
            output SD_M1PN : BOOL  // Digital Outputs - Byte 1.Output 12
            output SD_M2PN : BOOL  // Digital Outputs - Byte 1.Output 13
            output SD_M3PN : BOOL  // Digital Outputs - Byte 1.Output 14
            output SD_M4PN : BOOL  // Digital Outputs - Byte 1.Output 15
            output SD_LQUEI : BOOL  // Digital Outputs - Byte 1.Output 16
            output SD_MAIRLIF : BOOL  // Digital Outputs - Byte 1.Output 17
            unmapped channels: %QB10 Digital Outputs - Byte 0, %QB11 Digital Outputs - Byte 1
        NX2001_06 : NX2001, Altus S.A., order no. NX2001, version 1.2.0.10
            settings: Physical Address of the Slave = 261; DC sync0 cycletime = 4000; Diag Instance Id = 261; %Q Start Address of Module Diagnostics Area = 21568; Parameter list definition.Count = 16; Item_00000.Access Name.BaseType = 1; Item_00000.Access Name.Address = ADR(IoConfig_Globals_Mapping.SD_DUPAIRLIF); Item_00000.Access Name.SizeInBits = 1; Item_00000.Access Name.TotalSizeInBits = 1; Item_00001.Access Name.BaseType = 1; Item_00001.Access Name.Address = ADR(IoConfig_Globals_Mapping.SD_DUPTORRE); Item_00001.Access Name.BitOffset = 1; Item_00001.Access Name.SizeInBits = 1; Item_00001.Access Name.TotalSizeInBits = 1; Item_00002.Access Name.BaseType = 1; Item_00002.Access Name.Address = ADR(IoConfig_Globals_Mapping.SD_DUPATM); Item_00002.Access Name.BitOffset = 2; Item_00002.Access Name.SizeInBits = 1; Item_00002.Access Name.TotalSizeInBits = 1; Item_00003.Access Name.BaseType = 1; Item_00003.Access Name.Address = ADR(IoConfig_Globals_Mapping.SD_SONORO); Item_00003.Access Name.BitOffset = 3; Item_00003.Access Name.SizeInBits = 1; Item_00003.Access Name.TotalSizeInBits = 1; Item_00004.Access Name.BaseType = 1; Item_00004.Access Name.Address = ADR(IoConfig_Globals_Mapping.SD_Geral_ALAR); Item_00004.Access Name.BitOffset = 4; Item_00004.Access Name.SizeInBits = 1; Item_00004.Access Name.TotalSizeInBits = 1; Item_00005.Access Name.BaseType = 1; Item_00005.Access Name.Address = ADR(IoConfig_Globals_Mapping.SD_BLL2R); Item_00005.Access Name.BitOffset = 5; Item_00005.Access Name.SizeInBits = 1; Item_00005.Access Name.TotalSizeInBits = 1; Quality Variable Name.BaseType = 28; Quality Variable Name.Address = ADR(IOQualities.QUALITY_NX2001_06); Quality Variable Name.SizeInBits = 32; Quality Variable Name.TotalSizeInBits = 512
            output SD_DUPAIRLIF : BOOL  // Digital Outputs - Byte 0.Output 00
            output SD_DUPTORRE : BOOL  // Digital Outputs - Byte 0.Output 01
            output SD_DUPATM : BOOL  // Digital Outputs - Byte 0.Output 02
            output SD_SONORO : BOOL  // Digital Outputs - Byte 0.Output 03
            output SD_Geral_ALAR : BOOL  // Digital Outputs - Byte 0.Output 04
            output SD_BLL2R : BOOL  // Digital Outputs - Byte 0.Output 05
            unmapped channels: %QB12 Digital Outputs - Byte 0, %QB13 Digital Outputs - Byte 1
        NX1001 : NX1001, Altus S.A., order no. NX1001, version 1.2.0.10
            settings: Physical Address of the Slave = 4; DC sync0 cycletime = 4000; Diag Instance Id = 4; %Q Start Address of Module Diagnostics Area = 21572; Parameter list definition.Count = 16; Item_00000.Access Name.BaseType = 1; Item_00000.Access Name.Address = ADR(IoConfig_Globals_Mapping.ED_RPO1_L); Item_00000.Access Name.SizeInBits = 1; Item_00000.Access Name.TotalSizeInBits = 1; Item_00001.Access Name.BaseType = 1; Item_00001.Access Name.Address = ADR(IoConfig_Globals_Mapping.ED_RPO2_L); Item_00001.Access Name.BitOffset = 1; Item_00001.Access Name.SizeInBits = 1; Item_00001.Access Name.TotalSizeInBits = 1; Item_00002.Access Name.BaseType = 1; Item_00002.Access Name.Address = ADR(IoConfig_Globals_Mapping.ED_RPO3_L); Item_00002.Access Name.BitOffset = 2; Item_00002.Access Name.SizeInBits = 1; Item_00002.Access Name.TotalSizeInBits = 1; Item_00003.Access Name.BaseType = 1; Item_00003.Access Name.Address = ADR(IoConfig_Globals_Mapping.ED_RPO4_L); Item_00003.Access Name.BitOffset = 3; Item_00003.Access Name.SizeInBits = 1; Item_00003.Access Name.TotalSizeInBits = 1; Item_00004.Access Name.BaseType = 1; Item_00004.Access Name.Address = ADR(IoConfig_Globals_Mapping.ED_RPO5_L); Item_00004.Access Name.BitOffset = 4; Item_00004.Access Name.SizeInBits = 1; Item_00004.Access Name.TotalSizeInBits = 1; Item_00005.Access Name.BaseType = 1; Item_00005.Access Name.Address = ADR(IoConfig_Globals_Mapping.ED_RC6H_L); Item_00005.Access Name.BitOffset = 5; Item_00005.Access Name.SizeInBits = 1; Item_00005.Access Name.TotalSizeInBits = 1; Item_00006.Access Name.BaseType = 1; Item_00006.Access Name.Address = ADR(IoConfig_Globals_Mapping.ED_RC7I_L); Item_00006.Access Name.BitOffset = 6; Item_00006.Access Name.SizeInBits = 1; Item_00006.Access Name.TotalSizeInBits = 1; Item_00007.Access Name.BaseType = 1;
              Item_00007.Access Name.Address = ADR(IoConfig_Globals_Mapping.ED_BLS1D_L); Item_00007.Access Name.BitOffset = 7; Item_00007.Access Name.SizeInBits = 1; Item_00007.Access Name.TotalSizeInBits = 1; Item_00008.Access Name.BaseType = 1; Item_00008.Access Name.Address = ADR(IoConfig_Globals_Mapping.ED_BLS2D_L); Item_00008.Access Name.SizeInBits = 1; Item_00008.Access Name.TotalSizeInBits = 1; Item_00009.Access Name.BaseType = 1; Item_00009.Access Name.Address = ADR(IoConfig_Globals_Mapping.ED_BLS3D_L); Item_00009.Access Name.BitOffset = 1; Item_00009.Access Name.SizeInBits = 1; Item_00009.Access Name.TotalSizeInBits = 1; Item_00010.Access Name.BaseType = 1; Item_00010.Access Name.Address = ADR(IoConfig_Globals_Mapping.ED_BLS4D_L); Item_00010.Access Name.BitOffset = 2; Item_00010.Access Name.SizeInBits = 1; Item_00010.Access Name.TotalSizeInBits = 1; Item_00011.Access Name.BaseType = 1; Item_00011.Access Name.Address = ADR(IoConfig_Globals_Mapping.ED_BLS5D_L); Item_00011.Access Name.BitOffset = 3; Item_00011.Access Name.SizeInBits = 1; Item_00011.Access Name.TotalSizeInBits = 1; Item_00012.Access Name.BaseType = 1; Item_00012.Access Name.Address = ADR(IoConfig_Globals_Mapping.ED_BL1D_L); Item_00012.Access Name.BitOffset = 4; Item_00012.Access Name.SizeInBits = 1; Item_00012.Access Name.TotalSizeInBits = 1; Item_00013.Access Name.BaseType = 1; Item_00013.Access Name.Address = ADR(IoConfig_Globals_Mapping.ED_BL2D_L); Item_00013.Access Name.BitOffset = 5; Item_00013.Access Name.SizeInBits = 1; Item_00013.Access Name.TotalSizeInBits = 1; Item_00014.Access Name.BaseType = 1; Item_00014.Access Name.Address = ADR(IoConfig_Globals_Mapping.ED_BL3D_L); Item_00014.Access Name.BitOffset = 6; Item_00014.Access Name.SizeInBits = 1; Item_00014.Access Name.TotalSizeInBits = 1; Item_00015.Access Name.BaseType = 1; Item_00015.Access Name.Address = ADR(IoConfig_Globals_Mapping.ED_BL4D_L);
              Item_00015.Access Name.BitOffset = 7; Item_00015.Access Name.SizeInBits = 1; Item_00015.Access Name.TotalSizeInBits = 1; Quality Variable Name.BaseType = 28; Quality Variable Name.Address = ADR(IOQualities.QUALITY_NX1001); Quality Variable Name.SizeInBits = 32; Quality Variable Name.TotalSizeInBits = 512
            input  ED_RPO1_L : BOOL  // Digital Inputs - Byte 0.Input 00
            input  ED_RPO2_L : BOOL  // Digital Inputs - Byte 0.Input 01
            input  ED_RPO3_L : BOOL  // Digital Inputs - Byte 0.Input 02
            input  ED_RPO4_L : BOOL  // Digital Inputs - Byte 0.Input 03
            input  ED_RPO5_L : BOOL  // Digital Inputs - Byte 0.Input 04
            input  ED_RC6H_L : BOOL  // Digital Inputs - Byte 0.Input 05
            input  ED_RC7I_L : BOOL  // Digital Inputs - Byte 0.Input 06
            input  ED_BLS1D_L : BOOL  // Digital Inputs - Byte 0.Input 07
            input  ED_BLS2D_L : BOOL  // Digital Inputs - Byte 1.Input 10
            input  ED_BLS3D_L : BOOL  // Digital Inputs - Byte 1.Input 11
            input  ED_BLS4D_L : BOOL  // Digital Inputs - Byte 1.Input 12
            input  ED_BLS5D_L : BOOL  // Digital Inputs - Byte 1.Input 13
            input  ED_BL1D_L : BOOL  // Digital Inputs - Byte 1.Input 14
            input  ED_BL2D_L : BOOL  // Digital Inputs - Byte 1.Input 15
            input  ED_BL3D_L : BOOL  // Digital Inputs - Byte 1.Input 16
            input  ED_BL4D_L : BOOL  // Digital Inputs - Byte 1.Input 17
            unmapped channels: %IB0 Digital Inputs - Byte 0, %IB1 Digital Inputs - Byte 1
        NX1001_01 : NX1001, Altus S.A., order no. NX1001, version 1.2.0.10
            settings: Number of Outputs = 0; Number of Infos about Outputs = 0; Physical Address of the Slave = 5; Sync.FlagControl = 0; FMMU.EndBit = 0; FMMU.Flags = 0; DC sync0 cycletime = 4000; Diag Instance Id = 5; %Q Start Address of Module Diagnostics Area = 21574; Parameter list definition.Count = 16; Item_00000.Access Name.BaseType = 1; Item_00000.Access Name.Address = ADR(IoConfig_Globals_Mapping.ED_FLXAGUA); Item_00000.Access Name.SizeInBits = 1; Item_00000.Access Name.TotalSizeInBits = 1; Item_00001.Access Name.BaseType = 1; Item_00001.Access Name.Address = ADR(IoConfig_Globals_Mapping.ED_BLL1R_L); Item_00001.Access Name.BitOffset = 1; Item_00001.Access Name.SizeInBits = 1; Item_00001.Access Name.TotalSizeInBits = 1; Item_00002.Access Name.BaseType = 1; Item_00002.Access Name.Address = ADR(IoConfig_Globals_Mapping.ED_BLL1L_L); Item_00002.Access Name.BitOffset = 2; Item_00002.Access Name.SizeInBits = 1; Item_00002.Access Name.TotalSizeInBits = 1; Item_00003.Access Name.BaseType = 1; Item_00003.Access Name.Address = ADR(IoConfig_Globals_Mapping.ED_BLL2R_L); Item_00003.Access Name.BitOffset = 3; Item_00003.Access Name.SizeInBits = 1; Item_00003.Access Name.TotalSizeInBits = 1; Item_00004.Access Name.BaseType = 1; Item_00004.Access Name.Address = ADR(IoConfig_Globals_Mapping.ED_BLL2L_L); Item_00004.Access Name.BitOffset = 4; Item_00004.Access Name.SizeInBits = 1; Item_00004.Access Name.TotalSizeInBits = 1; Item_00005.Access Name.BaseType = 1; Item_00005.Access Name.Address = ADR(IoConfig_Globals_Mapping.ED_BLL3R_L); Item_00005.Access Name.BitOffset = 5; Item_00005.Access Name.SizeInBits = 1; Item_00005.Access Name.TotalSizeInBits = 1; Item_00006.Access Name.BaseType = 1;
              Item_00006.Access Name.Address = ADR(IoConfig_Globals_Mapping.ED_BLL3L_L); Item_00006.Access Name.BitOffset = 6; Item_00006.Access Name.SizeInBits = 1; Item_00006.Access Name.TotalSizeInBits = 1; Item_00007.Access Name.BaseType = 1; Item_00007.Access Name.Address = ADR(IoConfig_Globals_Mapping.ED_BLL4R_L); Item_00007.Access Name.BitOffset = 7; Item_00007.Access Name.SizeInBits = 1; Item_00007.Access Name.TotalSizeInBits = 1; Item_00008.Access Name.BaseType = 1; Item_00008.Access Name.Address = ADR(IoConfig_Globals_Mapping.ED_BLL4L_L); Item_00008.Access Name.SizeInBits = 1; Item_00008.Access Name.TotalSizeInBits = 1; Item_00009.Access Name.BaseType = 1; Item_00009.Access Name.Address = ADR(IoConfig_Globals_Mapping.ED_CFMXP_P); Item_00009.Access Name.BitOffset = 1; Item_00009.Access Name.SizeInBits = 1; Item_00009.Access Name.TotalSizeInBits = 1; Item_00010.Access Name.BaseType = 1; Item_00010.Access Name.Address = ADR(IoConfig_Globals_Mapping.ED_CFMXP_E); Item_00010.Access Name.BitOffset = 2; Item_00010.Access Name.SizeInBits = 1; Item_00010.Access Name.TotalSizeInBits = 1; Item_00011.Access Name.BaseType = 1; Item_00011.Access Name.Address = ADR(IoConfig_Globals_Mapping.ED_CFMXP_T); Item_00011.Access Name.BitOffset = 3; Item_00011.Access Name.SizeInBits = 1; Item_00011.Access Name.TotalSizeInBits = 1; Item_00012.Access Name.BaseType = 1; Item_00012.Access Name.Address = ADR(IoConfig_Globals_Mapping.ED_MXE); Item_00012.Access Name.BitOffset = 4; Item_00012.Access Name.SizeInBits = 1; Item_00012.Access Name.TotalSizeInBits = 1; Item_00013.Access Name.BaseType = 1; Item_00013.Access Name.Address = ADR(IoConfig_Globals_Mapping.ED_BOCOMB_L); Item_00013.Access Name.BitOffset = 5; Item_00013.Access Name.SizeInBits = 1; Item_00013.Access Name.TotalSizeInBits = 1; Item_00014.Access Name.BaseType = 1; Item_00014.Access Name.Address = ADR(IoConfig_Globals_Mapping.ED_BDP_L);
              Item_00014.Access Name.BitOffset = 6; Item_00014.Access Name.SizeInBits = 1; Item_00014.Access Name.TotalSizeInBits = 1; Item_00015.Access Name.BaseType = 1; Item_00015.Access Name.Address = ADR(IoConfig_Globals_Mapping.ED_BB_F); Item_00015.Access Name.BitOffset = 7; Item_00015.Access Name.SizeInBits = 1; Item_00015.Access Name.TotalSizeInBits = 1; Quality Variable Name.BaseType = 28; Quality Variable Name.Address = ADR(IOQualities.QUALITY_NX1001_01); Quality Variable Name.SizeInBits = 32; Quality Variable Name.TotalSizeInBits = 512
            input  ED_FLXAGUA : BOOL  // Digital Inputs - Byte 0.Input 00
            input  ED_BLL1R_L : BOOL  // Digital Inputs - Byte 0.Input 01
            input  ED_BLL1L_L : BOOL  // Digital Inputs - Byte 0.Input 02
            input  ED_BLL2R_L : BOOL  // Digital Inputs - Byte 0.Input 03
            input  ED_BLL2L_L : BOOL  // Digital Inputs - Byte 0.Input 04
            input  ED_BLL3R_L : BOOL  // Digital Inputs - Byte 0.Input 05
            input  ED_BLL3L_L : BOOL  // Digital Inputs - Byte 0.Input 06
            input  ED_BLL4R_L : BOOL  // Digital Inputs - Byte 0.Input 07
            input  ED_BLL4L_L : BOOL  // Digital Inputs - Byte 1.Input 10
            input  ED_CFMXP_P : BOOL  // Digital Inputs - Byte 1.Input 11
            input  ED_CFMXP_E : BOOL  // Digital Inputs - Byte 1.Input 12
            input  ED_CFMXP_T : BOOL  // Digital Inputs - Byte 1.Input 13
            input  ED_MXE : BOOL  // Digital Inputs - Byte 1.Input 14
            input  ED_BOCOMB_L : BOOL  // Digital Inputs - Byte 1.Input 15
            input  ED_BDP_L : BOOL  // Digital Inputs - Byte 1.Input 16
            input  ED_BB_F : BOOL  // Digital Inputs - Byte 1.Input 17
            unmapped channels: %IB2 Digital Inputs - Byte 0, %IB3 Digital Inputs - Byte 1
        NX1001_02 : NX1001, Altus S.A., order no. NX1001, version 1.2.0.10
            settings: Physical Address of the Slave = 6; DC sync0 cycletime = 4000; Diag Instance Id = 6; %Q Start Address of Module Diagnostics Area = 21576; Parameter list definition.Count = 16; Item_00000.Access Name.BaseType = 1; Item_00000.Access Name.Address = ADR(IoConfig_Globals_Mapping.ED_BA1_F); Item_00000.Access Name.SizeInBits = 1; Item_00000.Access Name.TotalSizeInBits = 1; Item_00001.Access Name.BaseType = 1; Item_00001.Access Name.Address = ADR(IoConfig_Globals_Mapping.ED_BA2_F); Item_00001.Access Name.BitOffset = 1; Item_00001.Access Name.SizeInBits = 1; Item_00001.Access Name.TotalSizeInBits = 1; Item_00002.Access Name.BaseType = 1; Item_00002.Access Name.Address = ADR(IoConfig_Globals_Mapping.ED_BA3_F); Item_00002.Access Name.BitOffset = 2; Item_00002.Access Name.SizeInBits = 1; Item_00002.Access Name.TotalSizeInBits = 1; Item_00003.Access Name.BaseType = 1; Item_00003.Access Name.Address = ADR(IoConfig_Globals_Mapping.ED_BSU_D); Item_00003.Access Name.BitOffset = 3; Item_00003.Access Name.SizeInBits = 1; Item_00003.Access Name.TotalSizeInBits = 1; Item_00004.Access Name.BaseType = 1; Item_00004.Access Name.Address = ADR(IoConfig_Globals_Mapping.ED_BSI_D); Item_00004.Access Name.BitOffset = 4; Item_00004.Access Name.SizeInBits = 1; Item_00004.Access Name.TotalSizeInBits = 1; Item_00005.Access Name.BaseType = 1; Item_00005.Access Name.Address = ADR(IoConfig_Globals_Mapping.ED_BA_D); Item_00005.Access Name.BitOffset = 5; Item_00005.Access Name.SizeInBits = 1; Item_00005.Access Name.TotalSizeInBits = 1; Item_00006.Access Name.BaseType = 1; Item_00006.Access Name.Address = ADR(IoConfig_Globals_Mapping.ED_BSO_D); Item_00006.Access Name.BitOffset = 6; Item_00006.Access Name.SizeInBits = 1; Item_00006.Access Name.TotalSizeInBits = 1; Item_00007.Access Name.BaseType = 1;
              Item_00007.Access Name.Address = ADR(IoConfig_Globals_Mapping.ED_BB_D); Item_00007.Access Name.BitOffset = 7; Item_00007.Access Name.SizeInBits = 1; Item_00007.Access Name.TotalSizeInBits = 1; Item_00008.Access Name.BaseType = 1; Item_00008.Access Name.Address = ADR(IoConfig_Globals_Mapping.ED_BTRA_D); Item_00008.Access Name.SizeInBits = 1; Item_00008.Access Name.TotalSizeInBits = 1; Item_00009.Access Name.BaseType = 1; Item_00009.Access Name.Address = ADR(IoConfig_Globals_Mapping.ED_BDP_D); Item_00009.Access Name.BitOffset = 1; Item_00009.Access Name.SizeInBits = 1; Item_00009.Access Name.TotalSizeInBits = 1; Item_00010.Access Name.BaseType = 1; Item_00010.Access Name.Address = ADR(IoConfig_Globals_Mapping.ED_BOCOMB_D); Item_00010.Access Name.BitOffset = 2; Item_00010.Access Name.SizeInBits = 1; Item_00010.Access Name.TotalSizeInBits = 1; Item_00011.Access Name.BaseType = 1; Item_00011.Access Name.Address = ADR(IoConfig_Globals_Mapping.ED_MTL_D); Item_00011.Access Name.BitOffset = 3; Item_00011.Access Name.SizeInBits = 1; Item_00011.Access Name.TotalSizeInBits = 1; Item_00012.Access Name.BaseType = 1; Item_00012.Access Name.Address = ADR(IoConfig_Globals_Mapping.ED_PRTBA1); Item_00012.Access Name.BitOffset = 4; Item_00012.Access Name.SizeInBits = 1; Item_00012.Access Name.TotalSizeInBits = 1; Item_00013.Access Name.BaseType = 1; Item_00013.Access Name.Address = ADR(IoConfig_Globals_Mapping.ED_PRTBA2); Item_00013.Access Name.BitOffset = 5; Item_00013.Access Name.SizeInBits = 1; Item_00013.Access Name.TotalSizeInBits = 1; Item_00014.Access Name.BaseType = 1; Item_00014.Access Name.Address = ADR(IoConfig_Globals_Mapping.ED_PRTMBTRANS); Item_00014.Access Name.BitOffset = 6; Item_00014.Access Name.SizeInBits = 1; Item_00014.Access Name.TotalSizeInBits = 1; Item_00015.Access Name.BaseType = 1; Item_00015.Access Name.Address = ADR(IoConfig_Globals_Mapping.ED_PRTLINHAALTA);
              Item_00015.Access Name.BitOffset = 7; Item_00015.Access Name.SizeInBits = 1; Item_00015.Access Name.TotalSizeInBits = 1; Quality Variable Name.BaseType = 28; Quality Variable Name.Address = ADR(IOQualities.QUALITY_NX1001_02); Quality Variable Name.SizeInBits = 32; Quality Variable Name.TotalSizeInBits = 512
            input  ED_BA1_F : BOOL  // Digital Inputs - Byte 0.Input 00
            input  ED_BA2_F : BOOL  // Digital Inputs - Byte 0.Input 01
            input  ED_BA3_F : BOOL  // Digital Inputs - Byte 0.Input 02
            input  ED_BSU_D : BOOL  // Digital Inputs - Byte 0.Input 03
            input  ED_BSI_D : BOOL  // Digital Inputs - Byte 0.Input 04
            input  ED_BA_D : BOOL  // Digital Inputs - Byte 0.Input 05
            input  ED_BSO_D : BOOL  // Digital Inputs - Byte 0.Input 06
            input  ED_BB_D : BOOL  // Digital Inputs - Byte 0.Input 07
            input  ED_BTRA_D : BOOL  // Digital Inputs - Byte 1.Input 10
            input  ED_BDP_D : BOOL  // Digital Inputs - Byte 1.Input 11
            input  ED_BOCOMB_D : BOOL  // Digital Inputs - Byte 1.Input 12
            input  ED_MTL_D : BOOL  // Digital Inputs - Byte 1.Input 13
            input  ED_PRTBA1 : BOOL  // Digital Inputs - Byte 1.Input 14
            input  ED_PRTBA2 : BOOL  // Digital Inputs - Byte 1.Input 15
            input  ED_PRTMBTRANS : BOOL  // Digital Inputs - Byte 1.Input 16
            input  ED_PRTLINHAALTA : BOOL  // Digital Inputs - Byte 1.Input 17
            unmapped channels: %IB4 Digital Inputs - Byte 0, %IB5 Digital Inputs - Byte 1
        NX4000 : NX4000, Altus S.A., order no. NX4000, version 1.1.0.12
            settings: Physical Address of the Slave = 14; DC sync0 cycletime = 4000; Diag Instance Id = 14; %Q Start Address of Module Diagnostics Area = 21578
            unmapped channels: Reserved
        NX8000_01 : NX8000, Altus S.A., order no. NX8000, version 1.0.1.4
            settings: Physical Address of the Slave = 256; DC sync0 cycletime = 4000; Diag Instance Id = 256
        NX1001_03 : NX1001, Altus S.A., order no. NX1001, version 1.2.0.10
            settings: Physical Address of the Slave = 7; DC sync0 cycletime = 4000; Diag Instance Id = 7; %Q Start Address of Module Diagnostics Area = 21590; Parameter list definition.Count = 16; Item_00000.Access Name.BaseType = 1; Item_00000.Access Name.Address = ADR(IoConfig_Globals_Mapping.BL_03_FLT); Item_00000.Access Name.SizeInBits = 1; Item_00000.Access Name.TotalSizeInBits = 1; Item_00001.Access Name.BaseType = 1; Item_00001.Access Name.Address = ADR(IoConfig_Globals_Mapping.BL_03_ST); Item_00001.Access Name.BitOffset = 1; Item_00001.Access Name.SizeInBits = 1; Item_00001.Access Name.TotalSizeInBits = 1; Item_00002.Access Name.BaseType = 1; Item_00002.Access Name.Address = ADR(IoConfig_Globals_Mapping.BA_03_PRESS); Item_00002.Access Name.BitOffset = 2; Item_00002.Access Name.SizeInBits = 1; Item_00002.Access Name.TotalSizeInBits = 1; Item_00003.Access Name.BaseType = 1; Item_00003.Access Name.Address = ADR(IoConfig_Globals_Mapping.ED_PNM1_L); Item_00003.Access Name.BitOffset = 3; Item_00003.Access Name.SizeInBits = 1; Item_00003.Access Name.TotalSizeInBits = 1; Item_00004.Access Name.BaseType = 1; Item_00004.Access Name.Address = ADR(IoConfig_Globals_Mapping.ED_PNM2_L); Item_00004.Access Name.BitOffset = 4; Item_00004.Access Name.SizeInBits = 1; Item_00004.Access Name.TotalSizeInBits = 1; Item_00005.Access Name.BaseType = 1; Item_00005.Access Name.Address = ADR(IoConfig_Globals_Mapping.ED_PNM3_L); Item_00005.Access Name.BitOffset = 5; Item_00005.Access Name.SizeInBits = 1; Item_00005.Access Name.TotalSizeInBits = 1; Item_00006.Access Name.BaseType = 1; Item_00006.Access Name.Address = ADR(IoConfig_Globals_Mapping.ED_PNM4_L); Item_00006.Access Name.BitOffset = 6; Item_00006.Access Name.SizeInBits = 1; Item_00006.Access Name.TotalSizeInBits = 1; Item_00007.Access Name.BaseType = 1;
              Item_00007.Access Name.Address = ADR(IoConfig_Globals_Mapping.ED_PNDMIX_L); Item_00007.Access Name.BitOffset = 7; Item_00007.Access Name.SizeInBits = 1; Item_00007.Access Name.TotalSizeInBits = 1; Item_00008.Access Name.BaseType = 1; Item_00008.Access Name.Address = ADR(IoConfig_Globals_Mapping.ED_CFEXFM1_P); Item_00008.Access Name.SizeInBits = 1; Item_00008.Access Name.TotalSizeInBits = 1; Item_00009.Access Name.BaseType = 1; Item_00009.Access Name.Address = ADR(IoConfig_Globals_Mapping.ED_CFEXFM1_E); Item_00009.Access Name.BitOffset = 1; Item_00009.Access Name.SizeInBits = 1; Item_00009.Access Name.TotalSizeInBits = 1; Item_00010.Access Name.BaseType = 1; Item_00010.Access Name.Address = ADR(IoConfig_Globals_Mapping.ED_CFEXFM1_T); Item_00010.Access Name.BitOffset = 2; Item_00010.Access Name.SizeInBits = 1; Item_00010.Access Name.TotalSizeInBits = 1; Item_00011.Access Name.BaseType = 1; Item_00011.Access Name.Address = ADR(IoConfig_Globals_Mapping.ED_CFEXFM2_P); Item_00011.Access Name.BitOffset = 3; Item_00011.Access Name.SizeInBits = 1; Item_00011.Access Name.TotalSizeInBits = 1; Item_00012.Access Name.BaseType = 1; Item_00012.Access Name.Address = ADR(IoConfig_Globals_Mapping.ED_CFEXFM2_E); Item_00012.Access Name.BitOffset = 4; Item_00012.Access Name.SizeInBits = 1; Item_00012.Access Name.TotalSizeInBits = 1; Item_00013.Access Name.BaseType = 1; Item_00013.Access Name.Address = ADR(IoConfig_Globals_Mapping.ED_CFEXFM2_T); Item_00013.Access Name.BitOffset = 5; Item_00013.Access Name.SizeInBits = 1; Item_00013.Access Name.TotalSizeInBits = 1; Item_00014.Access Name.BaseType = 1; Item_00014.Access Name.Address = ADR(IoConfig_Globals_Mapping.ED_EX125_ALAR); Item_00014.Access Name.BitOffset = 6; Item_00014.Access Name.SizeInBits = 1; Item_00014.Access Name.TotalSizeInBits = 1; Item_00015.Access Name.BaseType = 1; Item_00015.Access Name.Address = ADR(IoConfig_Globals_Mapping.ED_EX100_ALAR);
              Item_00015.Access Name.BitOffset = 7; Item_00015.Access Name.SizeInBits = 1; Item_00015.Access Name.TotalSizeInBits = 1; Quality Variable Name.BaseType = 28; Quality Variable Name.Address = ADR(IOQualities.QUALITY_NX1001_03); Quality Variable Name.SizeInBits = 32; Quality Variable Name.TotalSizeInBits = 512
            input  BL_03_FLT : BOOL  // Digital Inputs - Byte 0.Input 00
            input  BL_03_ST : BOOL  // Digital Inputs - Byte 0.Input 01
            input  BA_03_PRESS : BOOL  // Digital Inputs - Byte 0.Input 02
            input  ED_PNM1_L : BOOL  // Digital Inputs - Byte 0.Input 03
            input  ED_PNM2_L : BOOL  // Digital Inputs - Byte 0.Input 04
            input  ED_PNM3_L : BOOL  // Digital Inputs - Byte 0.Input 05
            input  ED_PNM4_L : BOOL  // Digital Inputs - Byte 0.Input 06
            input  ED_PNDMIX_L : BOOL  // Digital Inputs - Byte 0.Input 07
            input  ED_CFEXFM1_P : BOOL  // Digital Inputs - Byte 1.Input 10
            input  ED_CFEXFM1_E : BOOL  // Digital Inputs - Byte 1.Input 11
            input  ED_CFEXFM1_T : BOOL  // Digital Inputs - Byte 1.Input 12
            input  ED_CFEXFM2_P : BOOL  // Digital Inputs - Byte 1.Input 13
            input  ED_CFEXFM2_E : BOOL  // Digital Inputs - Byte 1.Input 14
            input  ED_CFEXFM2_T : BOOL  // Digital Inputs - Byte 1.Input 15
            input  ED_EX125_ALAR : BOOL  // Digital Inputs - Byte 1.Input 16
            input  ED_EX100_ALAR : BOOL  // Digital Inputs - Byte 1.Input 17
            unmapped channels: %IB7 Digital Inputs - Byte 0, %IB8 Digital Inputs - Byte 1
        NX1001_04 : NX1001, Altus S.A., order no. NX1001, version 1.2.0.10
            settings: Physical Address of the Slave = 8; DC sync0 cycletime = 4000; Diag Instance Id = 8; %Q Start Address of Module Diagnostics Area = 21592; Parameter list definition.Count = 16; Item_00000.Access Name.BaseType = 1; Item_00000.Access Name.Address = ADR(IoConfig_Globals_Mapping.ED_BP2); Item_00000.Access Name.SizeInBits = 1; Item_00000.Access Name.TotalSizeInBits = 1; Item_00001.Access Name.BaseType = 1; Item_00001.Access Name.Address = ADR(IoConfig_Globals_Mapping.ED_BP1); Item_00001.Access Name.BitOffset = 1; Item_00001.Access Name.SizeInBits = 1; Item_00001.Access Name.TotalSizeInBits = 1; Item_00002.Access Name.BaseType = 1; Item_00002.Access Name.Address = ADR(IoConfig_Globals_Mapping.ED_CFVEXFM2_P); Item_00002.Access Name.BitOffset = 2; Item_00002.Access Name.SizeInBits = 1; Item_00002.Access Name.TotalSizeInBits = 1; Item_00003.Access Name.BaseType = 1; Item_00003.Access Name.Address = ADR(IoConfig_Globals_Mapping.ED_CFVEXFM2_E); Item_00003.Access Name.BitOffset = 3; Item_00003.Access Name.SizeInBits = 1; Item_00003.Access Name.TotalSizeInBits = 1; Item_00004.Access Name.BaseType = 1; Item_00004.Access Name.Address = ADR(IoConfig_Globals_Mapping.ED_CFVEXFM2_T); Item_00004.Access Name.BitOffset = 4; Item_00004.Access Name.SizeInBits = 1; Item_00004.Access Name.TotalSizeInBits = 1; Item_00005.Access Name.BaseType = 1; Item_00005.Access Name.Address = ADR(IoConfig_Globals_Mapping.ED_VELAIRLF100); Item_00005.Access Name.BitOffset = 5; Item_00005.Access Name.SizeInBits = 1; Item_00005.Access Name.TotalSizeInBits = 1; Item_00006.Access Name.BaseType = 1; Item_00006.Access Name.Address = ADR(IoConfig_Globals_Mapping.ED_AIRLFT_F); Item_00006.Access Name.BitOffset = 6; Item_00006.Access Name.SizeInBits = 1; Item_00006.Access Name.TotalSizeInBits = 1; Item_00007.Access Name.BaseType = 1;
              Item_00007.Access Name.Address = ADR(IoConfig_Globals_Mapping.ED_DUPAIRLF_A); Item_00007.Access Name.BitOffset = 7; Item_00007.Access Name.SizeInBits = 1; Item_00007.Access Name.TotalSizeInBits = 1; Item_00008.Access Name.BaseType = 1; Item_00008.Access Name.Address = ADR(IoConfig_Globals_Mapping.ED_DUPAIRLF_F); Item_00008.Access Name.SizeInBits = 1; Item_00008.Access Name.TotalSizeInBits = 1; Item_00009.Access Name.BaseType = 1; Item_00009.Access Name.Address = ADR(IoConfig_Globals_Mapping.ED_DUPTORRE_F); Item_00009.Access Name.BitOffset = 1; Item_00009.Access Name.SizeInBits = 1; Item_00009.Access Name.TotalSizeInBits = 1; Item_00010.Access Name.BaseType = 1; Item_00010.Access Name.Address = ADR(IoConfig_Globals_Mapping.ED_DUPTORRE_A); Item_00010.Access Name.BitOffset = 2; Item_00010.Access Name.SizeInBits = 1; Item_00010.Access Name.TotalSizeInBits = 1; Item_00011.Access Name.BaseType = 1; Item_00011.Access Name.Address = ADR(IoConfig_Globals_Mapping.ED_DUPATM_F); Item_00011.Access Name.BitOffset = 3; Item_00011.Access Name.SizeInBits = 1; Item_00011.Access Name.TotalSizeInBits = 1; Item_00012.Access Name.BaseType = 1; Item_00012.Access Name.Address = ADR(IoConfig_Globals_Mapping.ED_DUPATM_A); Item_00012.Access Name.BitOffset = 4; Item_00012.Access Name.SizeInBits = 1; Item_00012.Access Name.TotalSizeInBits = 1; Item_00013.Access Name.BaseType = 1; Item_00013.Access Name.Address = ADR(IoConfig_Globals_Mapping.ED_DISJROSCADS07); Item_00013.Access Name.BitOffset = 5; Item_00013.Access Name.SizeInBits = 1; Item_00013.Access Name.TotalSizeInBits = 1; Item_00014.Access Name.BaseType = 1; Item_00014.Access Name.Address = ADR(IoConfig_Globals_Mapping.ED_PRESOCOMB); Item_00014.Access Name.BitOffset = 6; Item_00014.Access Name.SizeInBits = 1; Item_00014.Access Name.TotalSizeInBits = 1; Item_00015.Access Name.BaseType = 1; Item_00015.Access Name.Address = ADR(IoConfig_Globals_Mapping.ED_PRTMAXARCOM);
              Item_00015.Access Name.BitOffset = 7; Item_00015.Access Name.SizeInBits = 1; Item_00015.Access Name.TotalSizeInBits = 1; Quality Variable Name.BaseType = 28; Quality Variable Name.Address = ADR(IOQualities.QUALITY_NX1001_04); Quality Variable Name.SizeInBits = 32; Quality Variable Name.TotalSizeInBits = 512
            input  ED_BP2 : BOOL  // Digital Inputs - Byte 0.Input 00
            input  ED_BP1 : BOOL  // Digital Inputs - Byte 0.Input 01
            input  ED_CFVEXFM2_P : BOOL  // Digital Inputs - Byte 0.Input 02
            input  ED_CFVEXFM2_E : BOOL  // Digital Inputs - Byte 0.Input 03
            input  ED_CFVEXFM2_T : BOOL  // Digital Inputs - Byte 0.Input 04
            input  ED_VELAIRLF100 : BOOL  // Digital Inputs - Byte 0.Input 05
            input  ED_AIRLFT_F : BOOL  // Digital Inputs - Byte 0.Input 06
            input  ED_DUPAIRLF_A : BOOL  // Digital Inputs - Byte 0.Input 07
            input  ED_DUPAIRLF_F : BOOL  // Digital Inputs - Byte 1.Input 10
            input  ED_DUPTORRE_F : BOOL  // Digital Inputs - Byte 1.Input 11
            input  ED_DUPTORRE_A : BOOL  // Digital Inputs - Byte 1.Input 12
            input  ED_DUPATM_F : BOOL  // Digital Inputs - Byte 1.Input 13
            input  ED_DUPATM_A : BOOL  // Digital Inputs - Byte 1.Input 14
            input  ED_DISJROSCADS07 : BOOL  // Digital Inputs - Byte 1.Input 15
            input  ED_PRESOCOMB : BOOL  // Digital Inputs - Byte 1.Input 16
            input  ED_PRTMAXARCOM : BOOL  // Digital Inputs - Byte 1.Input 17
            unmapped channels: %IB9 Digital Inputs - Byte 0, %IB10 Digital Inputs - Byte 1
        NX1001_05 : NX1001, Altus S.A., order no. NX1001, version 1.2.0.10
            settings: Physical Address of the Slave = 9; DC sync0 cycletime = 4000; Diag Instance Id = 9; %Q Start Address of Module Diagnostics Area = 21594; Parameter list definition.Count = 16; Item_00000.Access Name.BaseType = 1; Item_00000.Access Name.Address = ADR(IoConfig_Globals_Mapping.ED_PRTMINARCOM); Item_00000.Access Name.SizeInBits = 1; Item_00000.Access Name.TotalSizeInBits = 1; Item_00001.Access Name.BaseType = 1; Item_00001.Access Name.Address = ADR(IoConfig_Globals_Mapping.ED_VLSMP_A); Item_00001.Access Name.BitOffset = 1; Item_00001.Access Name.SizeInBits = 1; Item_00001.Access Name.TotalSizeInBits = 1; Item_00002.Access Name.BaseType = 1; Item_00002.Access Name.Address = ADR(IoConfig_Globals_Mapping.ED_VLSMP_F); Item_00002.Access Name.BitOffset = 2; Item_00002.Access Name.SizeInBits = 1; Item_00002.Access Name.TotalSizeInBits = 1; Item_00003.Access Name.BaseType = 1; Item_00003.Access Name.Address = ADR(IoConfig_Globals_Mapping.ED_VLR_A); Item_00003.Access Name.BitOffset = 3; Item_00003.Access Name.SizeInBits = 1; Item_00003.Access Name.TotalSizeInBits = 1; Item_00004.Access Name.BaseType = 1; Item_00004.Access Name.Address = ADR(IoConfig_Globals_Mapping.ED_VLR_F); Item_00004.Access Name.BitOffset = 4; Item_00004.Access Name.SizeInBits = 1; Item_00004.Access Name.TotalSizeInBits = 1; Item_00005.Access Name.BaseType = 1; Item_00005.Access Name.Address = ADR(IoConfig_Globals_Mapping.ED_VLR_L); Item_00005.Access Name.BitOffset = 5; Item_00005.Access Name.SizeInBits = 1; Item_00005.Access Name.TotalSizeInBits = 1; Item_00006.Access Name.BaseType = 1; Item_00006.Access Name.Address = ADR(IoConfig_Globals_Mapping.ED_ESTST_L); Item_00006.Access Name.BitOffset = 6; Item_00006.Access Name.SizeInBits = 1; Item_00006.Access Name.TotalSizeInBits = 1; Item_00007.Access Name.BaseType = 1;
              Item_00007.Access Name.Address = ADR(IoConfig_Globals_Mapping.ED_ESTSAIRLF_L); Item_00007.Access Name.BitOffset = 7; Item_00007.Access Name.SizeInBits = 1; Item_00007.Access Name.TotalSizeInBits = 1; Item_00008.Access Name.BaseType = 1; Item_00008.Access Name.Address = ADR(IoConfig_Globals_Mapping.ED_TC3_L); Item_00008.Access Name.SizeInBits = 1; Item_00008.Access Name.TotalSizeInBits = 1; Item_00009.Access Name.BaseType = 1; Item_00009.Access Name.Address = ADR(IoConfig_Globals_Mapping.ED_ESTTC8_D); Item_00009.Access Name.BitOffset = 1; Item_00009.Access Name.SizeInBits = 1; Item_00009.Access Name.TotalSizeInBits = 1; Item_00010.Access Name.BaseType = 1; Item_00010.Access Name.Address = ADR(IoConfig_Globals_Mapping.ED_CFESTTC8_R); Item_00010.Access Name.BitOffset = 2; Item_00010.Access Name.SizeInBits = 1; Item_00010.Access Name.TotalSizeInBits = 1; Item_00011.Access Name.BaseType = 1; Item_00011.Access Name.Address = ADR(IoConfig_Globals_Mapping.ED_EL2_L); Item_00011.Access Name.BitOffset = 3; Item_00011.Access Name.SizeInBits = 1; Item_00011.Access Name.TotalSizeInBits = 1; Item_00012.Access Name.BaseType = 1; Item_00012.Access Name.Address = ADR(IoConfig_Globals_Mapping.ED_EL2_D); Item_00012.Access Name.BitOffset = 4; Item_00012.Access Name.SizeInBits = 1; Item_00012.Access Name.TotalSizeInBits = 1; Item_00013.Access Name.BaseType = 1; Item_00013.Access Name.Address = ADR(IoConfig_Globals_Mapping.ED_NVBO); Item_00013.Access Name.BitOffset = 5; Item_00013.Access Name.SizeInBits = 1; Item_00013.Access Name.TotalSizeInBits = 1; Item_00014.Access Name.BaseType = 1; Item_00014.Access Name.Address = ADR(IoConfig_Globals_Mapping.ED_NVAO); Item_00014.Access Name.BitOffset = 6; Item_00014.Access Name.SizeInBits = 1; Item_00014.Access Name.TotalSizeInBits = 1; Item_00015.Access Name.BaseType = 1; Item_00015.Access Name.Address = ADR(IoConfig_Globals_Mapping.ED_TM_OK);
              Item_00015.Access Name.BitOffset = 7; Item_00015.Access Name.SizeInBits = 1; Item_00015.Access Name.TotalSizeInBits = 1; Quality Variable Name.BaseType = 28; Quality Variable Name.Address = ADR(IOQualities.QUALITY_NX1001_05); Quality Variable Name.SizeInBits = 32; Quality Variable Name.TotalSizeInBits = 512
            input  ED_PRTMINARCOM : BOOL  // Digital Inputs - Byte 0.Input 00
            input  ED_VLSMP_A : BOOL  // Digital Inputs - Byte 0.Input 01
            input  ED_VLSMP_F : BOOL  // Digital Inputs - Byte 0.Input 02
            input  ED_VLR_A : BOOL  // Digital Inputs - Byte 0.Input 03
            input  ED_VLR_F : BOOL  // Digital Inputs - Byte 0.Input 04
            input  ED_VLR_L : BOOL  // Digital Inputs - Byte 0.Input 05
            input  ED_ESTST_L : BOOL  // Digital Inputs - Byte 0.Input 06
            input  ED_ESTSAIRLF_L : BOOL  // Digital Inputs - Byte 0.Input 07
            input  ED_TC3_L : BOOL  // Digital Inputs - Byte 1.Input 10
            input  ED_ESTTC8_D : BOOL  // Digital Inputs - Byte 1.Input 11
            input  ED_CFESTTC8_R : BOOL  // Digital Inputs - Byte 1.Input 12
            input  ED_EL2_L : BOOL  // Digital Inputs - Byte 1.Input 13
            input  ED_EL2_D : BOOL  // Digital Inputs - Byte 1.Input 14
            input  ED_NVBO : BOOL  // Digital Inputs - Byte 1.Input 15
            input  ED_NVAO : BOOL  // Digital Inputs - Byte 1.Input 16
            input  ED_TM_OK : BOOL  // Digital Inputs - Byte 1.Input 17
            unmapped channels: %IB11 Digital Inputs - Byte 0, %IB12 Digital Inputs - Byte 1
        NX1001_06 : NX1001, Altus S.A., order no. NX1001, version 1.2.0.10
            settings: Physical Address of the Slave = 10; DC sync0 cycletime = 4000; Diag Instance Id = 10; %Q Start Address of Module Diagnostics Area = 21596; Parameter list definition.Count = 16; Item_00000.Access Name.BaseType = 1; Item_00000.Access Name.Address = ADR(IoConfig_Globals_Mapping.ED_CHAFOR_A); Item_00000.Access Name.SizeInBits = 1; Item_00000.Access Name.TotalSizeInBits = 1; Item_00001.Access Name.BaseType = 1; Item_00001.Access Name.Address = ADR(IoConfig_Globals_Mapping.ED_PROGFOR_ALAR); Item_00001.Access Name.BitOffset = 1; Item_00001.Access Name.SizeInBits = 1; Item_00001.Access Name.TotalSizeInBits = 1; Item_00002.Access Name.BaseType = 1; Item_00002.Access Name.Address = ADR(IoConfig_Globals_Mapping.ED_PARREMLOC); Item_00002.Access Name.BitOffset = 2; Item_00002.Access Name.SizeInBits = 1; Item_00002.Access Name.TotalSizeInBits = 1; Item_00003.Access Name.BaseType = 1; Item_00003.Access Name.Address = ADR(IoConfig_Globals_Mapping.ED_BTEMER); Item_00003.Access Name.BitOffset = 3; Item_00003.Access Name.SizeInBits = 1; Item_00003.Access Name.TotalSizeInBits = 1; Item_00004.Access Name.BaseType = 1; Item_00004.Access Name.Address = ADR(IoConfig_Globals_Mapping.ED_FTF); Item_00004.Access Name.BitOffset = 4; Item_00004.Access Name.SizeInBits = 1; Item_00004.Access Name.TotalSizeInBits = 1; Item_00005.Access Name.BaseType = 1; Item_00005.Access Name.Address = ADR(IoConfig_Globals_Mapping.ED_MAXVL100); Item_00005.Access Name.BitOffset = 5; Item_00005.Access Name.SizeInBits = 1; Item_00005.Access Name.TotalSizeInBits = 1; Item_00006.Access Name.BaseType = 1; Item_00006.Access Name.Address = ADR(IoConfig_Globals_Mapping.ED_MINVL100); Item_00006.Access Name.BitOffset = 6; Item_00006.Access Name.SizeInBits = 1; Item_00006.Access Name.TotalSizeInBits = 1; Item_00007.Access Name.BaseType = 1;
              Item_00007.Access Name.Address = ADR(IoConfig_Globals_Mapping.CNT_L1); Item_00007.Access Name.BitOffset = 7; Item_00007.Access Name.SizeInBits = 1; Item_00007.Access Name.TotalSizeInBits = 1; Item_00008.Access Name.BaseType = 1; Item_00008.Access Name.Address = ADR(IoConfig_Globals_Mapping.CNT_L2); Item_00008.Access Name.SizeInBits = 1; Item_00008.Access Name.TotalSizeInBits = 1; Item_00009.Access Name.BaseType = 1; Item_00009.Access Name.Address = ADR(IoConfig_Globals_Mapping.CNT_L3); Item_00009.Access Name.BitOffset = 1; Item_00009.Access Name.SizeInBits = 1; Item_00009.Access Name.TotalSizeInBits = 1; Item_00010.Access Name.BaseType = 1; Item_00010.Access Name.Address = ADR(IoConfig_Globals_Mapping.CNT_L4); Item_00010.Access Name.BitOffset = 2; Item_00010.Access Name.SizeInBits = 1; Item_00010.Access Name.TotalSizeInBits = 1; Item_00011.Access Name.BaseType = 1; Item_00011.Access Name.Address = ADR(IoConfig_Globals_Mapping.CNT_L5); Item_00011.Access Name.BitOffset = 3; Item_00011.Access Name.SizeInBits = 1; Item_00011.Access Name.TotalSizeInBits = 1; Item_00012.Access Name.BaseType = 1; Item_00012.Access Name.Address = ADR(IoConfig_Globals_Mapping.CNT_L6); Item_00012.Access Name.BitOffset = 4; Item_00012.Access Name.SizeInBits = 1; Item_00012.Access Name.TotalSizeInBits = 1; Item_00013.Access Name.BaseType = 1; Item_00013.Access Name.Address = ADR(IoConfig_Globals_Mapping.CNT_L7); Item_00013.Access Name.BitOffset = 5; Item_00013.Access Name.SizeInBits = 1; Item_00013.Access Name.TotalSizeInBits = 1; Item_00014.Access Name.BaseType = 1; Item_00014.Access Name.Address = ADR(IoConfig_Globals_Mapping.CNT_L8); Item_00014.Access Name.BitOffset = 6; Item_00014.Access Name.SizeInBits = 1; Item_00014.Access Name.TotalSizeInBits = 1; Item_00015.Access Name.BaseType = 1; Item_00015.Access Name.Address = ADR(IoConfig_Globals_Mapping.CNT_L9);
              Item_00015.Access Name.BitOffset = 7; Item_00015.Access Name.SizeInBits = 1; Item_00015.Access Name.TotalSizeInBits = 1; Quality Variable Name.BaseType = 28; Quality Variable Name.Address = ADR(IOQualities.QUALITY_NX1001_06); Quality Variable Name.SizeInBits = 32; Quality Variable Name.TotalSizeInBits = 512
            input  ED_CHAFOR_A : BOOL  // Digital Inputs - Byte 0.Input 00
            input  ED_PROGFOR_ALAR : BOOL  // Digital Inputs - Byte 0.Input 01
            input  ED_PARREMLOC : BOOL  // Digital Inputs - Byte 0.Input 02
            input  ED_BTEMER : BOOL  // Digital Inputs - Byte 0.Input 03
            input  ED_FTF : BOOL  // Digital Inputs - Byte 0.Input 04
            input  ED_MAXVL100 : BOOL  // Digital Inputs - Byte 0.Input 05
            input  ED_MINVL100 : BOOL  // Digital Inputs - Byte 0.Input 06
            input  CNT_L1 : BOOL  // Digital Inputs - Byte 0.Input 07
            input  CNT_L2 : BOOL  // Digital Inputs - Byte 1.Input 10
            input  CNT_L3 : BOOL  // Digital Inputs - Byte 1.Input 11
            input  CNT_L4 : BOOL  // Digital Inputs - Byte 1.Input 12
            input  CNT_L5 : BOOL  // Digital Inputs - Byte 1.Input 13
            input  CNT_L6 : BOOL  // Digital Inputs - Byte 1.Input 14
            input  CNT_L7 : BOOL  // Digital Inputs - Byte 1.Input 15
            input  CNT_L8 : BOOL  // Digital Inputs - Byte 1.Input 16
            input  CNT_L9 : BOOL  // Digital Inputs - Byte 1.Input 17
            unmapped channels: %IB13 Digital Inputs - Byte 0, %IB14 Digital Inputs - Byte 1
        NX6000 : NX6000, Altus S.A., order no. NX6000, version 1.4.0.0
            settings: Physical Address of the Slave = 262; DC sync0 cycletime = 4000; Diag Instance Id = 262; %Q Start Address of Module Diagnostics Area = 21598; Parameter list definition.Count = 8; Item_00000.Access Name.BaseType = 7; Item_00000.Access Name.Address = ADR(IoConfig_Globals_Mapping.EA1); Item_00000.Access Name.SizeInBits = 16; Item_00000.Access Name.TotalSizeInBits = 16; Item_00001.Access Name.BaseType = 7; Item_00001.Access Name.Address = ADR(IoConfig_Globals_Mapping.EA2); Item_00001.Access Name.SizeInBits = 16; Item_00001.Access Name.TotalSizeInBits = 16; Item_00002.Access Name.BaseType = 7; Item_00002.Access Name.Address = ADR(IoConfig_Globals_Mapping.EA3); Item_00002.Access Name.SizeInBits = 16; Item_00002.Access Name.TotalSizeInBits = 16; Item_00003.Access Name.BaseType = 7; Item_00003.Access Name.Address = ADR(IoConfig_Globals_Mapping.EA4); Item_00003.Access Name.SizeInBits = 16; Item_00003.Access Name.TotalSizeInBits = 16; Item_00004.Access Name.BaseType = 7; Item_00004.Access Name.Address = ADR(IoConfig_Globals_Mapping.EA5); Item_00004.Access Name.SizeInBits = 16; Item_00004.Access Name.TotalSizeInBits = 16; Item_00005.Access Name.BaseType = 7; Item_00005.Access Name.Address = ADR(IoConfig_Globals_Mapping.EA6); Item_00005.Access Name.SizeInBits = 16; Item_00005.Access Name.TotalSizeInBits = 16; Item_00006.Access Name.BaseType = 7; Item_00006.Access Name.Address = ADR(IoConfig_Globals_Mapping.EA7); Item_00006.Access Name.SizeInBits = 16; Item_00006.Access Name.TotalSizeInBits = 16; Item_00007.Access Name.BaseType = 7; Item_00007.Access Name.Address = ADR(IoConfig_Globals_Mapping.EA8); Item_00007.Access Name.SizeInBits = 16; Item_00007.Access Name.TotalSizeInBits = 16; Quality Variable Name.BaseType = 28; Quality Variable Name.Address = ADR(IOQualities.QUALITY_NX6000); Quality Variable Name.SizeInBits = 32;
              Quality Variable Name.TotalSizeInBits = 256
            input  EA1 AT %IW15 : INT  // Analog Input 00
            input  EA2 AT %IW17 : INT  // Analog Input 01
            input  EA3 AT %IW19 : INT  // Analog Input 02
            input  EA4 AT %IW21 : INT  // Analog Input 03
            input  EA5 AT %IW23 : INT  // Analog Input 04
            input  EA6 AT %IW25 : INT  // Analog Input 05
            input  EA7 AT %IW27 : INT  // Analog Input 06
            input  EA8 AT %IW29 : INT  // Analog Input 07
        NX6000_01 : NX6000, Altus S.A., order no. NX6000, version 1.4.0.0
            settings: Physical Address of the Slave = 263; DC sync0 cycletime = 4000; Diag Instance Id = 263; %Q Start Address of Module Diagnostics Area = 21616; Parameter list definition.Count = 8; Item_00000.Access Name.BaseType = 7; Item_00000.Access Name.Address = ADR(IoConfig_Globals_Mapping.EA101); Item_00000.Access Name.SizeInBits = 16; Item_00000.Access Name.TotalSizeInBits = 16; Item_00001.Access Name.BaseType = 7; Item_00001.Access Name.Address = ADR(IoConfig_Globals_Mapping.EA201); Item_00001.Access Name.SizeInBits = 16; Item_00001.Access Name.TotalSizeInBits = 16; Item_00002.Access Name.BaseType = 7; Item_00002.Access Name.Address = ADR(IoConfig_Globals_Mapping.EA301); Item_00002.Access Name.SizeInBits = 16; Item_00002.Access Name.TotalSizeInBits = 16; Item_00003.Access Name.BaseType = 7; Item_00003.Access Name.Address = ADR(IoConfig_Globals_Mapping.EA401); Item_00003.Access Name.SizeInBits = 16; Item_00003.Access Name.TotalSizeInBits = 16; Item_00004.Access Name.BaseType = 7; Item_00004.Access Name.Address = ADR(IoConfig_Globals_Mapping.EA501); Item_00004.Access Name.SizeInBits = 16; Item_00004.Access Name.TotalSizeInBits = 16; Item_00005.Access Name.BaseType = 7; Item_00005.Access Name.Address = ADR(IoConfig_Globals_Mapping.EA601); Item_00005.Access Name.SizeInBits = 16; Item_00005.Access Name.TotalSizeInBits = 16; Item_00006.Access Name.BaseType = 7; Item_00006.Access Name.Address = ADR(IoConfig_Globals_Mapping.EA701); Item_00006.Access Name.SizeInBits = 16; Item_00006.Access Name.TotalSizeInBits = 16; Item_00007.Access Name.BaseType = 7; Item_00007.Access Name.Address = ADR(IoConfig_Globals_Mapping.EA801); Item_00007.Access Name.SizeInBits = 16; Item_00007.Access Name.TotalSizeInBits = 16; Quality Variable Name.BaseType = 28; Quality Variable Name.Address = ADR(IOQualities.QUALITY_NX6000_01); Quality Variable Name.SizeInBits = 32;
              Quality Variable Name.TotalSizeInBits = 256
            input  EA101 AT %IW31 : INT  // Analog Input 00
            input  EA201 AT %IW33 : INT  // Analog Input 01
            input  EA301 AT %IW35 : INT  // Analog Input 02
            input  EA401 AT %IW37 : INT  // Analog Input 03
            input  EA501 AT %IW39 : INT  // Analog Input 04
            input  EA601 AT %IW41 : INT  // Analog Input 05
            input  EA701 AT %IW43 : INT  // Analog Input 06
            input  EA801 AT %IW45 : INT  // Analog Input 07
        NX6000_02 : NX6000, Altus S.A., order no. NX6000, version 1.4.0.0
            settings: Physical Address of the Slave = 264; DC sync0 cycletime = 4000; Diag Instance Id = 264; %Q Start Address of Module Diagnostics Area = 21634; Parameter list definition.Count = 8; Item_00000.Access Name.BaseType = 7; Item_00000.Access Name.Address = ADR(IoConfig_Globals_Mapping.EA102); Item_00000.Access Name.SizeInBits = 16; Item_00000.Access Name.TotalSizeInBits = 16; Item_00001.Access Name.BaseType = 7; Item_00001.Access Name.Address = ADR(IoConfig_Globals_Mapping.EA202); Item_00001.Access Name.SizeInBits = 16; Item_00001.Access Name.TotalSizeInBits = 16; Item_00002.Access Name.BaseType = 7; Item_00002.Access Name.Address = ADR(IoConfig_Globals_Mapping.EA302); Item_00002.Access Name.SizeInBits = 16; Item_00002.Access Name.TotalSizeInBits = 16; Item_00003.Access Name.BaseType = 7; Item_00003.Access Name.Address = ADR(IoConfig_Globals_Mapping.EA402); Item_00003.Access Name.SizeInBits = 16; Item_00003.Access Name.TotalSizeInBits = 16; Item_00004.Access Name.BaseType = 7; Item_00004.Access Name.Address = ADR(IoConfig_Globals_Mapping.EA502); Item_00004.Access Name.SizeInBits = 16; Item_00004.Access Name.TotalSizeInBits = 16; Item_00005.Access Name.BaseType = 7; Item_00005.Access Name.Address = ADR(IoConfig_Globals_Mapping.EA602); Item_00005.Access Name.SizeInBits = 16; Item_00005.Access Name.TotalSizeInBits = 16; Item_00006.Access Name.BaseType = 7; Item_00006.Access Name.Address = ADR(IoConfig_Globals_Mapping.EA702); Item_00006.Access Name.SizeInBits = 16; Item_00006.Access Name.TotalSizeInBits = 16; Item_00007.Access Name.BaseType = 7; Item_00007.Access Name.Address = ADR(IoConfig_Globals_Mapping.EA802); Item_00007.Access Name.SizeInBits = 16; Item_00007.Access Name.TotalSizeInBits = 16; Quality Variable Name.BaseType = 28; Quality Variable Name.Address = ADR(IOQualities.QUALITY_NX6000_02); Quality Variable Name.SizeInBits = 32;
              Quality Variable Name.TotalSizeInBits = 256
            input  EA102 AT %IW47 : INT  // Analog Input 00
            input  EA202 AT %IW49 : INT  // Analog Input 01
            input  EA302 AT %IW51 : INT  // Analog Input 02
            input  EA402 AT %IW53 : INT  // Analog Input 03
            input  EA502 AT %IW55 : INT  // Analog Input 04
            input  EA602 AT %IW57 : INT  // Analog Input 05
            input  EA702 AT %IW59 : INT  // Analog Input 06
            input  EA802 AT %IW61 : INT  // Analog Input 07
        NX6010 : NX6010, Altus S.A., order no. NX6010, version 1.0.0.12
            settings: Physical Address of the Slave = 265; DC sync0 cycletime = 4000; Diag Instance Id = 265; %Q Start Address of Module Diagnostics Area = 21652; Parameter list definition.Count = 8; Item_00000.Access Name.BaseType = 7; Item_00000.Access Name.Address = ADR(IoConfig_Globals_Mapping.TEMPVAPOR); Item_00000.Access Name.SizeInBits = 16; Item_00000.Access Name.TotalSizeInBits = 16; Item_00002.Access Name.BaseType = 7; Item_00002.Access Name.Address = ADR(IoConfig_Globals_Mapping.TEMPQUEIMATORRE); Item_00002.Access Name.SizeInBits = 16; Item_00002.Access Name.TotalSizeInBits = 16; Item_00003.Access Name.BaseType = 7; Item_00003.Access Name.Address = ADR(IoConfig_Globals_Mapping.TEMPQUEIMADORATM); Item_00003.Access Name.SizeInBits = 16; Item_00003.Access Name.TotalSizeInBits = 16; Item_00004.Access Name.BaseType = 7; Item_00004.Access Name.Address = ADR(IoConfig_Globals_Mapping.TEMPTORE); Item_00004.Access Name.SizeInBits = 16; Item_00004.Access Name.TotalSizeInBits = 16; Quality Variable Name.BaseType = 28; Quality Variable Name.Address = ADR(IOQualities.QUALITY_NX6010); Quality Variable Name.SizeInBits = 32; Quality Variable Name.TotalSizeInBits = 256
            input  TEMPVAPOR AT %IW63 : INT  // Analog Input 00
            input  TEMPQUEIMATORRE AT %IW67 : INT  // Analog Input 02
            input  TEMPQUEIMADORATM AT %IW69 : INT  // Analog Input 03
            input  TEMPTORE AT %IW71 : INT  // Analog Input 04
            unmapped channels: %IW65 Analog Input 01, %IW73 Analog Input 05, %IW75 Analog Input 06, %IW77 Analog Input 07
        NX6100 : NX6100, Altus S.A., order no. NX6100, version 1.2.0.10
            settings: Physical Address of the Slave = 266; DC sync0 cycletime = 4000; Diag Instance Id = 266; %Q Start Address of Module Diagnostics Area = 21670; Parameter list definition.Count = 4; Item_00000.Access Name.BaseType = 7; Item_00000.Access Name.Address = ADR(IoConfig_Globals_Mapping.SA1); Item_00000.Access Name.SizeInBits = 16; Item_00000.Access Name.TotalSizeInBits = 16; Item_00001.Access Name.BaseType = 7; Item_00001.Access Name.Address = ADR(IoConfig_Globals_Mapping.SA2); Item_00001.Access Name.SizeInBits = 16; Item_00001.Access Name.TotalSizeInBits = 16; Item_00002.Access Name.BaseType = 7; Item_00002.Access Name.Address = ADR(IoConfig_Globals_Mapping.SA3); Item_00002.Access Name.SizeInBits = 16; Item_00002.Access Name.TotalSizeInBits = 16; Item_00003.Access Name.BaseType = 7; Item_00003.Access Name.Address = ADR(IoConfig_Globals_Mapping.SA4); Item_00003.Access Name.SizeInBits = 16; Item_00003.Access Name.TotalSizeInBits = 16; Quality Variable Name.BaseType = 28; Quality Variable Name.Address = ADR(IOQualities.QUALITY_NX6100); Quality Variable Name.SizeInBits = 32; Quality Variable Name.TotalSizeInBits = 128
            output SA1 AT %QW14 : INT  // Analog Output 00
            output SA2 AT %QW16 : INT  // Analog Output 01
            output SA3 AT %QW18 : INT  // Analog Output 02
            output SA4 AT %QW20 : INT  // Analog Output 03
        NX6100_01 : NX6100, Altus S.A., order no. NX6100, version 1.2.0.10
            settings: Physical Address of the Slave = 267; DC sync0 cycletime = 4000; Diag Instance Id = 267; %Q Start Address of Module Diagnostics Area = 21680; Parameter list definition.Count = 4; Item_00000.Access Name.BaseType = 7; Item_00000.Access Name.Address = ADR(IoConfig_Globals_Mapping.SA101); Item_00000.Access Name.SizeInBits = 16; Item_00000.Access Name.TotalSizeInBits = 16; Item_00001.Access Name.BaseType = 7; Item_00001.Access Name.Address = ADR(IoConfig_Globals_Mapping.SA201); Item_00001.Access Name.SizeInBits = 16; Item_00001.Access Name.TotalSizeInBits = 16; Item_00002.Access Name.BaseType = 7; Item_00002.Access Name.Address = ADR(IoConfig_Globals_Mapping.SA301); Item_00002.Access Name.SizeInBits = 16; Item_00002.Access Name.TotalSizeInBits = 16; Item_00003.Access Name.BaseType = 7; Item_00003.Access Name.Address = ADR(IoConfig_Globals_Mapping.SA401); Item_00003.Access Name.SizeInBits = 16; Item_00003.Access Name.TotalSizeInBits = 16; Quality Variable Name.BaseType = 28; Quality Variable Name.Address = ADR(IOQualities.QUALITY_NX6100_01); Quality Variable Name.SizeInBits = 32; Quality Variable Name.TotalSizeInBits = 128
            output SA101 AT %QW22 : INT  // Analog Output 00
            output SA201 AT %QW24 : INT  // Analog Output 01
            output SA301 AT %QW26 : INT  // Analog Output 02
            output SA401 AT %QW28 : INT  // Analog Output 03
        NX6100_02 : NX6100, Altus S.A., order no. NX6100, version 1.2.0.10
            settings: Physical Address of the Slave = 268; DC sync0 cycletime = 4000; Diag Instance Id = 268; %Q Start Address of Module Diagnostics Area = 21690; Parameter list definition.Count = 4; Item_00000.Access Name.BaseType = 7; Item_00000.Access Name.Address = ADR(IoConfig_Globals_Mapping.SA102); Item_00000.Access Name.SizeInBits = 16; Item_00000.Access Name.TotalSizeInBits = 16; Item_00001.Access Name.BaseType = 7; Item_00001.Access Name.Address = ADR(IoConfig_Globals_Mapping.SA202); Item_00001.Access Name.SizeInBits = 16; Item_00001.Access Name.TotalSizeInBits = 16; Item_00002.Access Name.BaseType = 7; Item_00002.Access Name.Address = ADR(IoConfig_Globals_Mapping.SA302); Item_00002.Access Name.SizeInBits = 16; Item_00002.Access Name.TotalSizeInBits = 16; Item_00003.Access Name.BaseType = 7; Item_00003.Access Name.Address = ADR(IoConfig_Globals_Mapping.SA402); Item_00003.Access Name.SizeInBits = 16; Item_00003.Access Name.TotalSizeInBits = 16; Quality Variable Name.BaseType = 28; Quality Variable Name.Address = ADR(IOQualities.QUALITY_NX6100_02); Quality Variable Name.SizeInBits = 32; Quality Variable Name.TotalSizeInBits = 128
            output SA102 AT %QW30 : INT  // Analog Output 00
            output SA202 AT %QW32 : INT  // Analog Output 01
            output SA302 AT %QW34 : INT  // Analog Output 02
            output SA402 AT %QW36 : INT  // Analog Output 03
        NX4000_01 : NX4000, Altus S.A., order no. NX4000, version 1.1.0.12
            settings: Physical Address of the Slave = 270; DC sync0 cycletime = 4000; Diag Instance Id = 270; %Q Start Address of Module Diagnostics Area = 21700
            unmapped channels: Reserved
        NX6000_03 : NX6000, Altus S.A., order no. NX6000, version 1.4.0.0
            settings: Physical Address of the Slave = 269; DC sync0 cycletime = 4000; Diag Instance Id = 269; %Q Start Address of Module Diagnostics Area = 23558; Parameter list definition.Count = 8; Item_00000.Access Name.BaseType = 7; Item_00000.Access Name.Address = ADR(IoConfig_Globals_Mapping.EA103); Item_00000.Access Name.SizeInBits = 16; Item_00000.Access Name.TotalSizeInBits = 16; Item_00001.Access Name.BaseType = 7; Item_00001.Access Name.Address = ADR(IoConfig_Globals_Mapping.EA203); Item_00001.Access Name.SizeInBits = 16; Item_00001.Access Name.TotalSizeInBits = 16; Item_00002.Access Name.BaseType = 7; Item_00002.Access Name.Address = ADR(IoConfig_Globals_Mapping.EA303); Item_00002.Access Name.SizeInBits = 16; Item_00002.Access Name.TotalSizeInBits = 16; Item_00003.Access Name.BaseType = 7; Item_00003.Access Name.Address = ADR(IoConfig_Globals_Mapping.EA403); Item_00003.Access Name.SizeInBits = 16; Item_00003.Access Name.TotalSizeInBits = 16; Item_00004.Access Name.BaseType = 7; Item_00004.Access Name.Address = ADR(IoConfig_Globals_Mapping.EA503); Item_00004.Access Name.SizeInBits = 16; Item_00004.Access Name.TotalSizeInBits = 16; Item_00005.Access Name.BaseType = 7; Item_00005.Access Name.Address = ADR(IoConfig_Globals_Mapping.EA603); Item_00005.Access Name.SizeInBits = 16; Item_00005.Access Name.TotalSizeInBits = 16; Item_00006.Access Name.BaseType = 7; Item_00006.Access Name.Address = ADR(IoConfig_Globals_Mapping.EA703); Item_00006.Access Name.SizeInBits = 16; Item_00006.Access Name.TotalSizeInBits = 16; Item_00007.Access Name.BaseType = 7; Item_00007.Access Name.Address = ADR(IoConfig_Globals_Mapping.EA803); Item_00007.Access Name.SizeInBits = 16; Item_00007.Access Name.TotalSizeInBits = 16; Quality Variable Name.BaseType = 28; Quality Variable Name.Address = ADR(IOQualities.QUALITY_NX6000_03); Quality Variable Name.SizeInBits = 32;
              Quality Variable Name.TotalSizeInBits = 256
            input  EA103 AT %IW80 : INT  // Analog Input 00
            input  EA203 AT %IW82 : INT  // Analog Input 01
            input  EA303 AT %IW84 : INT  // Analog Input 02
            input  EA403 AT %IW86 : INT  // Analog Input 03
            input  EA503 AT %IW88 : INT  // Analog Input 04
            input  EA603 AT %IW90 : INT  // Analog Input 05
            input  EA703 AT %IW92 : INT  // Analog Input 06
            input  EA803 AT %IW94 : INT  // Analog Input 07
  program ProdL8 [ST]
*)

// Device/Application/Diagnostics
VAR_GLOBAL
	//DG_MODBUS_Symbol_Client diagnostics variable
	DG_MODBUS_Symbol_Client              : T_DIAG_MODBUS_ETH_CLIENT_1;
	//DG_NX2001 diagnostics variable
	DG_NX2001                AT %QB21544 : T_DIAG_NX2001_1;
	//DG_NX2001_01 diagnostics variable
	DG_NX2001_01             AT %QB21548 : T_DIAG_NX2001_1;
	//DG_NX2001_02 diagnostics variable
	DG_NX2001_02             AT %QB21552 : T_DIAG_NX2001_1;
	//DG_NX2001_03 diagnostics variable
	DG_NX2001_03             AT %QB21556 : T_DIAG_NX2001_1;
	//DG_NX2001_04 diagnostics variable
	DG_NX2001_04             AT %QB21560 : T_DIAG_NX2001_1;
	//DG_NX2001_05 diagnostics variable
	DG_NX2001_05             AT %QB21564 : T_DIAG_NX2001_1;
	//DG_NX2001_06 diagnostics variable
	DG_NX2001_06             AT %QB21568 : T_DIAG_NX2001_1;
	//DG_NX1001 diagnostics variable
	DG_NX1001                AT %QB21572 : T_DIAG_NX1001_1;
	//DG_NX1001_01 diagnostics variable
	DG_NX1001_01             AT %QB21574 : T_DIAG_NX1001_1;
	//DG_NX1001_02 diagnostics variable
	DG_NX1001_02             AT %QB21576 : T_DIAG_NX1001_1;
	//DG_NX4000 diagnostics variable
	DG_NX4000                AT %QB21578 : T_DIAG_NX4000_1;
	//DG_NX1001_03 diagnostics variable
	DG_NX1001_03             AT %QB21590 : T_DIAG_NX1001_1;
	//DG_NX1001_04 diagnostics variable
	DG_NX1001_04             AT %QB21592 : T_DIAG_NX1001_1;
	//DG_NX1001_05 diagnostics variable
	DG_NX1001_05             AT %QB21594 : T_DIAG_NX1001_1;
	//DG_NX1001_06 diagnostics variable
	DG_NX1001_06             AT %QB21596 : T_DIAG_NX1001_1;
	//DG_NX6000 diagnostics variable
	DG_NX6000                AT %QB21598 : T_DIAG_NX6000_1;
	//DG_NX6000_01 diagnostics variable
	DG_NX6000_01             AT %QB21616 : T_DIAG_NX6000_1;
	//DG_NX6000_02 diagnostics variable
	DG_NX6000_02             AT %QB21634 : T_DIAG_NX6000_1;
	//DG_NX6010 diagnostics variable
	DG_NX6010                AT %QB21652 : T_DIAG_NX6010_1;
	//DG_NX6100 diagnostics variable
	DG_NX6100                AT %QB21670 : T_DIAG_NX6100_1;
	//DG_NX6100_01 diagnostics variable
	DG_NX6100_01             AT %QB21680 : T_DIAG_NX6100_1;
	//DG_NX6100_02 diagnostics variable
	DG_NX6100_02             AT %QB21690 : T_DIAG_NX6100_1;
	//DG_NX4000_01 diagnostics variable
	DG_NX4000_01             AT %QB21700 : T_DIAG_NX4000_1;
	//DG_MODBUS_Server diagnostics variable
	DG_MODBUS_Server         AT %QB21712 : T_DIAG_MODBUS_ETH_SERVER_1;
	//DG_MODBUS_RTU_Master diagnostics variable
	DG_MODBUS_RTU_Master     AT %QB21732 : T_DIAG_MODBUS_RTU_MASTER_1;
	//DG_Dosador1_Mapping_000 diagnostics variable
	DG_Dosador1_Mapping_000  AT %QB21752 : T_DIAG_MODBUS_RTU_MAPPING_1;
	//DG_Dosador1_Mapping_001 diagnostics variable
	DG_Dosador1_Mapping_001  AT %QB21760 : T_DIAG_MODBUS_RTU_MAPPING_1;
	//DG_Dosador1_Mapping_002 diagnostics variable
	DG_Dosador1_Mapping_002  AT %QB21768 : T_DIAG_MODBUS_RTU_MAPPING_1;
	//DG_Dosador1_Mapping_003 diagnostics variable
	DG_Dosador1_Mapping_003  AT %QB21776 : T_DIAG_MODBUS_RTU_MAPPING_1;
	//DG_Dosador1_Mapping_004 diagnostics variable
	DG_Dosador1_Mapping_004  AT %QB21784 : T_DIAG_MODBUS_RTU_MAPPING_1;
	//DG_Dosador1_Mapping_005 diagnostics variable
	DG_Dosador1_Mapping_005  AT %QB21792 : T_DIAG_MODBUS_RTU_MAPPING_1;
	//DG_Dosador1_Mapping_006 diagnostics variable
	DG_Dosador1_Mapping_006  AT %QB21800 : T_DIAG_MODBUS_RTU_MAPPING_1;
	//DG_Dosador2_Mapping_000 diagnostics variable
	DG_Dosador2_Mapping_000  AT %QB21808 : T_DIAG_MODBUS_RTU_MAPPING_1;
	//DG_Dosador2_Mapping_001 diagnostics variable
	DG_Dosador2_Mapping_001  AT %QB21816 : T_DIAG_MODBUS_RTU_MAPPING_1;
	//DG_Dosador2_Mapping_002 diagnostics variable
	DG_Dosador2_Mapping_002  AT %QB21824 : T_DIAG_MODBUS_RTU_MAPPING_1;
	//DG_Dosador2_Mapping_003 diagnostics variable
	DG_Dosador2_Mapping_003  AT %QB21832 : T_DIAG_MODBUS_RTU_MAPPING_1;
	//DG_Dosador2_Mapping_004 diagnostics variable
	DG_Dosador2_Mapping_004  AT %QB21840 : T_DIAG_MODBUS_RTU_MAPPING_1;
	//DG_Dosador2_Mapping_005 diagnostics variable
	DG_Dosador2_Mapping_005  AT %QB21848 : T_DIAG_MODBUS_RTU_MAPPING_1;
	//DG_Dosador2_Mapping_006 diagnostics variable
	DG_Dosador2_Mapping_006  AT %QB21856 : T_DIAG_MODBUS_RTU_MAPPING_1;
	//DG_Dosador3_Mapping_000 diagnostics variable
	DG_Dosador3_Mapping_000  AT %QB21864 : T_DIAG_MODBUS_RTU_MAPPING_1;
	//DG_Dosador3_Mapping_001 diagnostics variable
	DG_Dosador3_Mapping_001  AT %QB21872 : T_DIAG_MODBUS_RTU_MAPPING_1;
	//DG_Dosador3_Mapping_002 diagnostics variable
	DG_Dosador3_Mapping_002  AT %QB21880 : T_DIAG_MODBUS_RTU_MAPPING_1;
	//DG_Dosador3_Mapping_003 diagnostics variable
	DG_Dosador3_Mapping_003  AT %QB21888 : T_DIAG_MODBUS_RTU_MAPPING_1;
	//DG_Dosador3_Mapping_004 diagnostics variable
	DG_Dosador3_Mapping_004  AT %QB21896 : T_DIAG_MODBUS_RTU_MAPPING_1;
	//DG_Dosador3_Mapping_005 diagnostics variable
	DG_Dosador3_Mapping_005  AT %QB21904 : T_DIAG_MODBUS_RTU_MAPPING_1;
	//DG_Dosador3_Mapping_006 diagnostics variable
	DG_Dosador3_Mapping_006  AT %QB21912 : T_DIAG_MODBUS_RTU_MAPPING_1;
	//DG_Dosador4_Mapping_000 diagnostics variable
	DG_Dosador4_Mapping_000  AT %QB21920 : T_DIAG_MODBUS_RTU_MAPPING_1;
	//DG_Dosador4_Mapping_001 diagnostics variable
	DG_Dosador4_Mapping_001  AT %QB21928 : T_DIAG_MODBUS_RTU_MAPPING_1;
	//DG_Dosador4_Mapping_002 diagnostics variable
	DG_Dosador4_Mapping_002  AT %QB21936 : T_DIAG_MODBUS_RTU_MAPPING_1;
	//DG_Dosador4_Mapping_003 diagnostics variable
	DG_Dosador4_Mapping_003  AT %QB21944 : T_DIAG_MODBUS_RTU_MAPPING_1;
	//DG_Dosador4_Mapping_004 diagnostics variable
	DG_Dosador4_Mapping_004  AT %QB21952 : T_DIAG_MODBUS_RTU_MAPPING_1;
	//DG_Dosador4_Mapping_005 diagnostics variable
	DG_Dosador4_Mapping_005  AT %QB21960 : T_DIAG_MODBUS_RTU_MAPPING_1;
	//DG_Dosador4_Mapping_006 diagnostics variable
	DG_Dosador4_Mapping_006  AT %QB21968 : T_DIAG_MODBUS_RTU_MAPPING_1;
	//DG_Dosador5_Mapping_000 diagnostics variable
	DG_Dosador5_Mapping_000  AT %QB21976 : T_DIAG_MODBUS_RTU_MAPPING_1;
	//DG_Dosador5_Mapping_001 diagnostics variable
	DG_Dosador5_Mapping_001  AT %QB21984 : T_DIAG_MODBUS_RTU_MAPPING_1;
	//DG_Dosador5_Mapping_002 diagnostics variable
	DG_Dosador5_Mapping_002  AT %QB21992 : T_DIAG_MODBUS_RTU_MAPPING_1;
	//DG_Dosador5_Mapping_003 diagnostics variable
	DG_Dosador5_Mapping_003  AT %QB22000 : T_DIAG_MODBUS_RTU_MAPPING_1;
	//DG_Dosador5_Mapping_004 diagnostics variable
	DG_Dosador5_Mapping_004  AT %QB22008 : T_DIAG_MODBUS_RTU_MAPPING_1;
	//DG_Dosador5_Mapping_005 diagnostics variable
	DG_Dosador5_Mapping_005  AT %QB22016 : T_DIAG_MODBUS_RTU_MAPPING_1;
	//DG_Dosador5_Mapping_006 diagnostics variable
	DG_Dosador5_Mapping_006  AT %QB22024 : T_DIAG_MODBUS_RTU_MAPPING_1;
	//DG_Dosador7_Mapping_000 diagnostics variable
	DG_Dosador7_Mapping_000  AT %QB22032 : T_DIAG_MODBUS_RTU_MAPPING_1;
	//DG_Dosador7_Mapping_001 diagnostics variable
	DG_Dosador7_Mapping_001  AT %QB22040 : T_DIAG_MODBUS_RTU_MAPPING_1;
	//DG_Dosador7_Mapping_002 diagnostics variable
	DG_Dosador7_Mapping_002  AT %QB22048 : T_DIAG_MODBUS_RTU_MAPPING_1;
	//DG_Dosador7_Mapping_003 diagnostics variable
	DG_Dosador7_Mapping_003  AT %QB22056 : T_DIAG_MODBUS_RTU_MAPPING_1;
	//DG_Dosador7_Mapping_004 diagnostics variable
	DG_Dosador7_Mapping_004  AT %QB22064 : T_DIAG_MODBUS_RTU_MAPPING_1;
	//DG_Dosador7_Mapping_005 diagnostics variable
	DG_Dosador7_Mapping_005  AT %QB22072 : T_DIAG_MODBUS_RTU_MAPPING_1;
	//DG_Dosador7_Mapping_006 diagnostics variable
	DG_Dosador7_Mapping_006  AT %QB22080 : T_DIAG_MODBUS_RTU_MAPPING_1;
	//DG_Dosador8_Mapping_000 diagnostics variable
	DG_Dosador8_Mapping_000  AT %QB22088 : T_DIAG_MODBUS_RTU_MAPPING_1;
	//DG_Dosador8_Mapping_001 diagnostics variable
	DG_Dosador8_Mapping_001  AT %QB22096 : T_DIAG_MODBUS_RTU_MAPPING_1;
	//DG_Dosador8_Mapping_002 diagnostics variable
	DG_Dosador8_Mapping_002  AT %QB22104 : T_DIAG_MODBUS_RTU_MAPPING_1;
	//DG_Dosador8_Mapping_003 diagnostics variable
	DG_Dosador8_Mapping_003  AT %QB22112 : T_DIAG_MODBUS_RTU_MAPPING_1;
	//DG_Dosador8_Mapping_004 diagnostics variable
	DG_Dosador8_Mapping_004  AT %QB22120 : T_DIAG_MODBUS_RTU_MAPPING_1;
	//DG_Dosador8_Mapping_005 diagnostics variable
	DG_Dosador8_Mapping_005  AT %QB22128 : T_DIAG_MODBUS_RTU_MAPPING_1;
	//DG_Dosador8_Mapping_006 diagnostics variable
	DG_Dosador8_Mapping_006  AT %QB22136 : T_DIAG_MODBUS_RTU_MAPPING_1;
	//DG_Dosador9_Mapping_000 diagnostics variable
	DG_Dosador9_Mapping_000  AT %QB22144 : T_DIAG_MODBUS_RTU_MAPPING_1;
	//DG_Dosador9_Mapping_001 diagnostics variable
	DG_Dosador9_Mapping_001  AT %QB22152 : T_DIAG_MODBUS_RTU_MAPPING_1;
	//DG_Dosador9_Mapping_002 diagnostics variable
	DG_Dosador9_Mapping_002  AT %QB22160 : T_DIAG_MODBUS_RTU_MAPPING_1;
	//DG_Dosador9_Mapping_003 diagnostics variable
	DG_Dosador9_Mapping_003  AT %QB22168 : T_DIAG_MODBUS_RTU_MAPPING_1;
	//DG_Dosador9_Mapping_004 diagnostics variable
	DG_Dosador9_Mapping_004  AT %QB22176 : T_DIAG_MODBUS_RTU_MAPPING_1;
	//DG_Dosador9_Mapping_005 diagnostics variable
	DG_Dosador9_Mapping_005  AT %QB22184 : T_DIAG_MODBUS_RTU_MAPPING_1;
	//DG_Dosador9_Mapping_006 diagnostics variable
	DG_Dosador9_Mapping_006  AT %QB22192 : T_DIAG_MODBUS_RTU_MAPPING_1;
	//DG_Dosador10_Mapping_000 diagnostics variable
	DG_Dosador10_Mapping_000 AT %QB22200 : T_DIAG_MODBUS_RTU_MAPPING_1;
	//DG_Dosador10_Mapping_001 diagnostics variable
	DG_Dosador10_Mapping_001 AT %QB22208 : T_DIAG_MODBUS_RTU_MAPPING_1;
	//DG_Dosador10_Mapping_002 diagnostics variable
	DG_Dosador10_Mapping_002 AT %QB22216 : T_DIAG_MODBUS_RTU_MAPPING_1;
	//DG_Dosador10_Mapping_003 diagnostics variable
	DG_Dosador10_Mapping_003 AT %QB22224 : T_DIAG_MODBUS_RTU_MAPPING_1;
	//DG_Dosador10_Mapping_004 diagnostics variable
	DG_Dosador10_Mapping_004 AT %QB22232 : T_DIAG_MODBUS_RTU_MAPPING_1;
	//DG_Dosador10_Mapping_005 diagnostics variable
	DG_Dosador10_Mapping_005 AT %QB22240 : T_DIAG_MODBUS_RTU_MAPPING_1;
	//DG_Dosador10_Mapping_006 diagnostics variable
	DG_Dosador10_Mapping_006 AT %QB22248 : T_DIAG_MODBUS_RTU_MAPPING_1;
	//DG_Dosador11_Mapping_000 diagnostics variable
	DG_Dosador11_Mapping_000 AT %QB22256 : T_DIAG_MODBUS_RTU_MAPPING_1;
	//DG_Dosador11_Mapping_001 diagnostics variable
	DG_Dosador11_Mapping_001 AT %QB22264 : T_DIAG_MODBUS_RTU_MAPPING_1;
	//DG_Dosador11_Mapping_002 diagnostics variable
	DG_Dosador11_Mapping_002 AT %QB22272 : T_DIAG_MODBUS_RTU_MAPPING_1;
	//DG_Dosador11_Mapping_003 diagnostics variable
	DG_Dosador11_Mapping_003 AT %QB22280 : T_DIAG_MODBUS_RTU_MAPPING_1;
	//DG_Dosador11_Mapping_004 diagnostics variable
	DG_Dosador11_Mapping_004 AT %QB22288 : T_DIAG_MODBUS_RTU_MAPPING_1;
	//DG_Dosador11_Mapping_005 diagnostics variable
	DG_Dosador11_Mapping_005 AT %QB22296 : T_DIAG_MODBUS_RTU_MAPPING_1;
	//DG_Dosador11_Mapping_006 diagnostics variable
	DG_Dosador11_Mapping_006 AT %QB22304 : T_DIAG_MODBUS_RTU_MAPPING_1;
	//DG_Dosador12_Mapping_000 diagnostics variable
	DG_Dosador12_Mapping_000 AT %QB22312 : T_DIAG_MODBUS_RTU_MAPPING_1;
	//DG_Dosador12_Mapping_001 diagnostics variable
	DG_Dosador12_Mapping_001 AT %QB22320 : T_DIAG_MODBUS_RTU_MAPPING_1;
	//DG_Dosador12_Mapping_002 diagnostics variable
	DG_Dosador12_Mapping_002 AT %QB22328 : T_DIAG_MODBUS_RTU_MAPPING_1;
	//DG_Dosador12_Mapping_003 diagnostics variable
	DG_Dosador12_Mapping_003 AT %QB22336 : T_DIAG_MODBUS_RTU_MAPPING_1;
	//DG_Dosador12_Mapping_004 diagnostics variable
	DG_Dosador12_Mapping_004 AT %QB22344 : T_DIAG_MODBUS_RTU_MAPPING_1;
	//DG_Dosador12_Mapping_005 diagnostics variable
	DG_Dosador12_Mapping_005 AT %QB22352 : T_DIAG_MODBUS_RTU_MAPPING_1;
	//DG_Dosador12_Mapping_006 diagnostics variable
	DG_Dosador12_Mapping_006 AT %QB22360 : T_DIAG_MODBUS_RTU_MAPPING_1;
	//DG_Dosador13_Mapping_000 diagnostics variable
	DG_Dosador13_Mapping_000 AT %QB22368 : T_DIAG_MODBUS_RTU_MAPPING_1;
	//DG_Dosador13_Mapping_001 diagnostics variable
	DG_Dosador13_Mapping_001 AT %QB22376 : T_DIAG_MODBUS_RTU_MAPPING_1;
	//DG_Dosador13_Mapping_002 diagnostics variable
	DG_Dosador13_Mapping_002 AT %QB22384 : T_DIAG_MODBUS_RTU_MAPPING_1;
	//DG_Dosador13_Mapping_003 diagnostics variable
	DG_Dosador13_Mapping_003 AT %QB22392 : T_DIAG_MODBUS_RTU_MAPPING_1;
	//DG_Dosador13_Mapping_004 diagnostics variable
	DG_Dosador13_Mapping_004 AT %QB22400 : T_DIAG_MODBUS_RTU_MAPPING_1;
	//DG_Dosador13_Mapping_005 diagnostics variable
	DG_Dosador13_Mapping_005 AT %QB22408 : T_DIAG_MODBUS_RTU_MAPPING_1;
	//DG_Dosador13_Mapping_006 diagnostics variable
	DG_Dosador13_Mapping_006 AT %QB22416 : T_DIAG_MODBUS_RTU_MAPPING_1;
	//DG_Dosador1_Mapping_007 diagnostics variable
	DG_Dosador1_Mapping_007  AT %QB22424 : T_DIAG_MODBUS_RTU_MAPPING_1;
	//DG_Dosador1_Mapping_008 diagnostics variable
	DG_Dosador1_Mapping_008  AT %QB22432 : T_DIAG_MODBUS_RTU_MAPPING_1;
	//DG_Dosador1_Mapping_009 diagnostics variable
	DG_Dosador1_Mapping_009  AT %QB22440 : T_DIAG_MODBUS_RTU_MAPPING_1;
	//DG_Dosador2_Mapping_007 diagnostics variable
	DG_Dosador2_Mapping_007  AT %QB22448 : T_DIAG_MODBUS_RTU_MAPPING_1;
	//DG_Dosador2_Mapping_008 diagnostics variable
	DG_Dosador2_Mapping_008  AT %QB22456 : T_DIAG_MODBUS_RTU_MAPPING_1;
	//DG_Dosador2_Mapping_009 diagnostics variable
	DG_Dosador2_Mapping_009  AT %QB22464 : T_DIAG_MODBUS_RTU_MAPPING_1;
	//DG_Dosador3_Mapping_007 diagnostics variable
	DG_Dosador3_Mapping_007  AT %QB22472 : T_DIAG_MODBUS_RTU_MAPPING_1;
	//DG_Dosador3_Mapping_008 diagnostics variable
	DG_Dosador3_Mapping_008  AT %QB22480 : T_DIAG_MODBUS_RTU_MAPPING_1;
	//DG_Dosador3_Mapping_009 diagnostics variable
	DG_Dosador3_Mapping_009  AT %QB22488 : T_DIAG_MODBUS_RTU_MAPPING_1;
	//DG_Dosador4_Mapping_007 diagnostics variable
	DG_Dosador4_Mapping_007  AT %QB22496 : T_DIAG_MODBUS_RTU_MAPPING_1;
	//DG_Dosador4_Mapping_008 diagnostics variable
	DG_Dosador4_Mapping_008  AT %QB22504 : T_DIAG_MODBUS_RTU_MAPPING_1;
	//DG_Dosador4_Mapping_009 diagnostics variable
	DG_Dosador4_Mapping_009  AT %QB22512 : T_DIAG_MODBUS_RTU_MAPPING_1;
	//DG_Dosador5_Mapping_007 diagnostics variable
	DG_Dosador5_Mapping_007  AT %QB22520 : T_DIAG_MODBUS_RTU_MAPPING_1;
	//DG_Dosador5_Mapping_008 diagnostics variable
	DG_Dosador5_Mapping_008  AT %QB22528 : T_DIAG_MODBUS_RTU_MAPPING_1;
	//DG_Dosador5_Mapping_009 diagnostics variable
	DG_Dosador5_Mapping_009  AT %QB22536 : T_DIAG_MODBUS_RTU_MAPPING_1;
	//DG_Dosador7_Mapping_007 diagnostics variable
	DG_Dosador7_Mapping_007  AT %QB22544 : T_DIAG_MODBUS_RTU_MAPPING_1;
	//DG_Dosador7_Mapping_008 diagnostics variable
	DG_Dosador7_Mapping_008  AT %QB22552 : T_DIAG_MODBUS_RTU_MAPPING_1;
	//DG_Dosador7_Mapping_009 diagnostics variable
	DG_Dosador7_Mapping_009  AT %QB22560 : T_DIAG_MODBUS_RTU_MAPPING_1;
	//DG_Dosador8_Mapping_007 diagnostics variable
	DG_Dosador8_Mapping_007  AT %QB22568 : T_DIAG_MODBUS_RTU_MAPPING_1;
	//DG_Dosador8_Mapping_008 diagnostics variable
	DG_Dosador8_Mapping_008  AT %QB22576 : T_DIAG_MODBUS_RTU_MAPPING_1;
	//DG_Dosador8_Mapping_009 diagnostics variable
	DG_Dosador8_Mapping_009  AT %QB22584 : T_DIAG_MODBUS_RTU_MAPPING_1;
	//DG_Dosador9_Mapping_007 diagnostics variable
	DG_Dosador9_Mapping_007  AT %QB22592 : T_DIAG_MODBUS_RTU_MAPPING_1;
	//DG_Dosador9_Mapping_008 diagnostics variable
	DG_Dosador9_Mapping_008  AT %QB22600 : T_DIAG_MODBUS_RTU_MAPPING_1;
	//DG_Dosador9_Mapping_009 diagnostics variable
	DG_Dosador9_Mapping_009  AT %QB22608 : T_DIAG_MODBUS_RTU_MAPPING_1;
	//DG_Dosador10_Mapping_007 diagnostics variable
	DG_Dosador10_Mapping_007 AT %QB22616 : T_DIAG_MODBUS_RTU_MAPPING_1;
	//DG_Dosador10_Mapping_008 diagnostics variable
	DG_Dosador10_Mapping_008 AT %QB22624 : T_DIAG_MODBUS_RTU_MAPPING_1;
	//DG_Dosador10_Mapping_009 diagnostics variable
	DG_Dosador10_Mapping_009 AT %QB22632 : T_DIAG_MODBUS_RTU_MAPPING_1;
	//DG_Dosador11_Mapping_007 diagnostics variable
	DG_Dosador11_Mapping_007 AT %QB22640 : T_DIAG_MODBUS_RTU_MAPPING_1;
	//DG_Dosador11_Mapping_008 diagnostics variable
	DG_Dosador11_Mapping_008 AT %QB22648 : T_DIAG_MODBUS_RTU_MAPPING_1;
	//DG_Dosador11_Mapping_009 diagnostics variable
	DG_Dosador11_Mapping_009 AT %QB22656 : T_DIAG_MODBUS_RTU_MAPPING_1;
	//DG_Dosador12_Mapping_007 diagnostics variable
	DG_Dosador12_Mapping_007 AT %QB22664 : T_DIAG_MODBUS_RTU_MAPPING_1;
	//DG_Dosador12_Mapping_008 diagnostics variable
	DG_Dosador12_Mapping_008 AT %QB22672 : T_DIAG_MODBUS_RTU_MAPPING_1;
	//DG_Dosador12_Mapping_009 diagnostics variable
	DG_Dosador12_Mapping_009 AT %QB22680 : T_DIAG_MODBUS_RTU_MAPPING_1;
	//DG_Dosador13_Mapping_007 diagnostics variable
	DG_Dosador13_Mapping_007 AT %QB22688 : T_DIAG_MODBUS_RTU_MAPPING_1;
	//DG_Dosador13_Mapping_008 diagnostics variable
	DG_Dosador13_Mapping_008 AT %QB22696 : T_DIAG_MODBUS_RTU_MAPPING_1;
	//DG_Dosador13_Mapping_009 diagnostics variable
	DG_Dosador13_Mapping_009 AT %QB22704 : T_DIAG_MODBUS_RTU_MAPPING_1;
	//DG_NX3010 diagnostics variable
	DG_NX3010                AT %QB23000 : T_DIAG_NX3010_1;
	//DG_NX6000_03 diagnostics variable
	DG_NX6000_03             AT %QB23558 : T_DIAG_NX6000_1;
	//DG_Dosador14_Mapping_001 diagnostics variable
	DG_Dosador14_Mapping_001 AT %QB23584 : T_DIAG_MODBUS_RTU_MAPPING_1;
	//DG_Dosador14_Mapping_000 diagnostics variable
	DG_Dosador14_Mapping_000 AT %QB23592 : T_DIAG_MODBUS_RTU_MAPPING_1;
	//DG_Dosador14_Mapping_002 diagnostics variable
	DG_Dosador14_Mapping_002 AT %QB23600 : T_DIAG_MODBUS_RTU_MAPPING_1;
	//DG_Dosador14_Mapping_006 diagnostics variable
	DG_Dosador14_Mapping_006 AT %QB23632 : T_DIAG_MODBUS_RTU_MAPPING_1;
	//DG_Dosador14_Mapping_007 diagnostics variable
	DG_Dosador14_Mapping_007 AT %QB23640 : T_DIAG_MODBUS_RTU_MAPPING_1;
	//DG_Dosador14_Mapping_008 diagnostics variable
	DG_Dosador14_Mapping_008 AT %QB23648 : T_DIAG_MODBUS_RTU_MAPPING_1;
	//DG_Dosador14_Mapping_009 diagnostics variable
	DG_Dosador14_Mapping_009 AT %QB23656 : T_DIAG_MODBUS_RTU_MAPPING_1;
END_VAR

// Device/Application/GVLStatus
//Global Variable List de status dos equipamentos
VAR_GLOBAL
	
	//Status Mexedor principal ligado
	ST_CFMXP AT %QX3103.0:BOOL;		
	//Ciclo em processo
	ST_CICLO_PROCESSO AT %QX3105.6:BOOL;
	
	//WORD - bloco 1 de status
	Status1 AT %QW3120:WORD;
	//WORD - bloco 2 de status
	Status2 AT %QW3122:WORD;
	//WORD - bloco 3 de status
	Status3 AT %QW3124:WORD;
	//WORD - bloco 4 de status
	Status4 AT %QW3126:WORD;
	//WORD - bloco 5 de status
	Status5 AT %QW3128:WORD;
	//WORD - bloco 6 de status
	Status6 AT %QW3130:WORD;
	//WORD - bloco 7 de status
	Status7 AT %QW3132:WORD;

END_VAR

// Device/Application/GVLAlarmes
//Global Variable List de alarmes dos equipamentos
VAR_GLOBAL
	
